KUKA KRL program: MyProgram_277().src

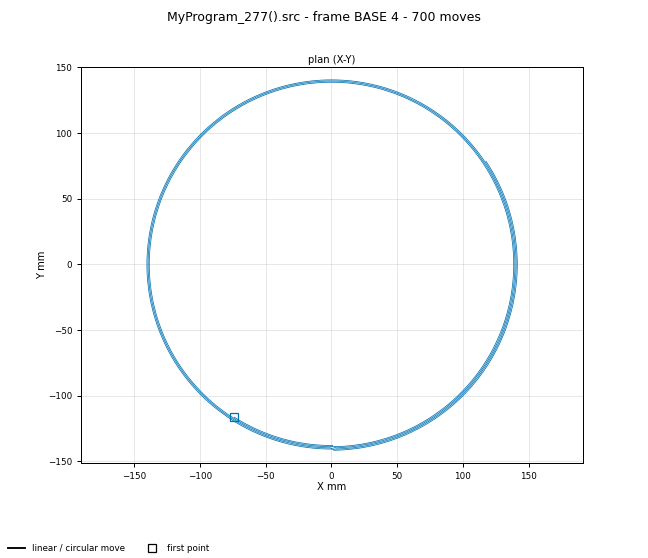
[picture p0: tool path of MyProgram_277().src in frame BASE 4, 700 of 700 moves have a stored position in this frame; points joined in program order, loops and branches not executed]
&ACCESS RVP
&REL 1
&PARAM TEMPLATE = C:\KRC\Roboter\Template\vorgabe
&PARAM EDITMASK = *
DEF MyProgram_277()
; ---- Setting reference (Base) ----
$BASE = BASE_DATA[4]

; --------------------------
; ---- Setting tool (TCP) ----
$TOOL = TOOL_DATA[3]
; --------------------------

$VEL.CP = VEL_APROX_PRINT
Startdeposition()
$VEL.CP = VEL_PRINT
LIN {X -74.0204,Y -116.2499,Z 172,A -119.7118,B 8.7917,C 0.3604,E1 8.715,E2 211.1655} C_DIS
LIN {X -70.2915,Y -118.5418,Z 172,A -117.8625,B 8.7917,C 0.3625,E1 8.7194,E2 209.3126} C_DIS
LIN {X -66.8151,Y -120.535,Z 172,A -115.8663,B 8.7917,C 0.3586,E1 8.7244,E2 207.2739} C_DIS
LIN {X -63.5094,Y -122.3084,Z 172,A -114.6724,B 8.7914,C 0.3673,E1 8.7272,E2 206.1271} C_DIS
LIN {X -60.8141,Y -123.6692,Z 172,A -113.4023,B 8.7914,C 0.3685,E1 8.7304,E2 204.8552} C_DIS
LIN {X -57.5799,Y -125.208,Z 172,A -111.8385,B 8.7914,C 0.3688,E1 8.7344,E2 203.2817} C_DIS
LIN {X -53.8139,Y -126.8742,Z 172,A -110.2313,B 8.7912,C 0.3725,E1 8.7385,E2 201.6879} C_DIS
LIN {X -51.2665,Y -127.9227,Z 172,A -109.0577,B 8.7912,C 0.3731,E1 8.7415,E2 200.5105} C_DIS
LIN {X -48.1192,Y -129.1395,Z 172,A -107.6615,B 8.7912,C 0.3745,E1 8.7452,E2 199.115} C_DIS
LIN {X -44.9658,Y -130.271,Z 172,A -106.2334,B 8.7912,C 0.375,E1 8.7489,E2 197.6822} C_DIS
LIN {X -41.408,Y -131.4462,Z 172,A -104.7037,B 8.791,C 0.3768,E1 8.753,E2 196.1559} C_DIS
LIN {X -38.8546,Y -132.2225,Z 172,A -103.5654,B 8.791,C 0.377,E1 8.7561,E2 195.0136} C_DIS
LIN {X -35.5653,Y -133.1449,Z 172,A -101.6158,B 8.7914,C 0.3678,E1 8.7615,E2 192.9952} C_DIS
LIN {X -31.1537,Y -134.2466,Z 172,A -100.099,B 8.7911,C 0.376,E1 8.7655,E2 191.5264} C_DIS
LIN {X -27.2255,Y -135.0974,Z 172,A -98.5166,B 8.791,C 0.3785,E1 8.7698,E2 189.9551} C_DIS
LIN {X -20.3148,Y -136.31,Z 172,A -95.7036,B 8.7908,C 0.3816,E1 8.7775,E2 187.1547} C_DIS
LIN {X -15.2753,Y -136.9652,Z 172,A -93.6377,B 8.7908,C 0.383,E1 8.7832,E2 185.0941} C_DIS
LIN {X -10.9275,Y -137.3811,Z 172,A -91.725,B 8.7908,C 0.3814,E1 8.7886,E2 183.1682} C_DIS
LIN {X -6.9698,Y -137.6371,Z 172,A -90.0219,B 8.7908,C 0.3804,E1 8.7933,E2 181.4573} C_DIS
LIN {X -2.6982,Y -137.7877,Z 172,A -88.2523,B 8.7908,C 0.3804,E1 8.7983,E2 179.688} C_DIS
LIN {X 0.9964,Y -137.8086,Z 172,A -86.8036,B 8.7908,C 0.382,E1 8.8023,E2 178.2498} C_DIS
Enddeposition()
LIN {X 0.9964,Y -137.8086,Z 172,A -86.8036,B 8.7908,C 0.382,E1 8.8023,E2 178.2498} C_DIS
Startdeposition()
$VEL.CP = VEL_PRINT
LIN {X 0.3242,Y -138.723,Z 172,A -87.6639,B 8.7185,C 0.4,E1 8.7281,E2 179.2402} C_DIS
LIN {X -3.8469,Y -138.6693,Z 172,A -89.329,B 8.7185,C 0.399,E1 8.7235,E2 180.8986} C_DIS
LIN {X -7.4248,Y -138.5245,Z 172,A -90.8807,B 8.7185,C 0.4004,E1 8.7191,E2 182.4603} C_DIS
LIN {X -11.8596,Y -138.2148,Z 172,A -92.6356,B 8.7185,C 0.3986,E1 8.7142,E2 184.2055} C_DIS
LIN {X -15.7064,Y -137.8324,Z 172,A -94.3982,B 8.7185,C 0.4015,E1 8.7093,E2 185.9901} C_DIS
LIN {X -20.165,Y -137.2501,Z 172,A -96.04,B 8.7187,C 0.3969,E1 8.7048,E2 187.6048} C_DIS
LIN {X -25.2134,Y -136.4125,Z 172,A -98.1321,B 8.7187,C 0.3957,E1 8.6991,E2 189.6948} C_DIS
LIN {X -28.3715,Y -135.792,Z 172,A -100.7545,B 8.7176,C 0.4193,E1 8.6915,E2 192.4824} C_DIS
LIN {X -36.4566,Y -133.8481,Z 172,A -102.9549,B 8.7188,C 0.3943,E1 8.6859,E2 194.5266} C_DIS
LIN {X -40.684,Y -132.6223,Z 172,A -104.8022,B 8.7188,C 0.3935,E1 8.681,E2 196.378} C_DIS
LIN {X -44.116,Y -131.5208,Z 172,A -106.2938,B 8.7188,C 0.3924,E1 8.677,E2 197.8702} C_DIS
LIN {X -47.3205,Y -130.402,Z 172,A -107.7112,B 8.7189,C 0.3915,E1 8.6733,E2 199.2898} C_DIS
LIN {X -50.4841,Y -129.2101,Z 172,A -109.1546,B 8.7189,C 0.3911,E1 8.6695,E2 200.7394} C_DIS
LIN {X -54.4235,Y -127.6024,Z 172,A -111.1054,B 8.7189,C 0.3928,E1 8.6644,E2 202.7151} C_DIS
LIN {X -58.4565,Y -125.8042,Z 172,A -112.7486,B 8.7191,C 0.3876,E1 8.6603,E2 204.3352} C_DIS
LIN {X -61.9898,Y -124.1029,Z 172,A -115.1913,B 8.7185,C 0.4004,E1 8.6539,E2 206.8828} C_DIS
LIN {X -67.5425,Y -121.1715,Z 172,A -117.0477,B 8.7192,C 0.384,E1 8.6496,E2 208.6456} C_DIS
LIN {X -71.4012,Y -118.9387,Z 172,A -118.9419,B 8.7193,C 0.3824,E1 8.645,E2 210.5464} C_DIS
LIN {X -75.2542,Y -116.5388,Z 172,A -120.8416,B 8.7194,C 0.3801,E1 8.6405,E2 212.4491} C_DIS
LIN {X -79.0577,Y -113.9925,Z 172,A -122.7073,B 8.7195,C 0.3767,E1 8.6362,E2 214.3114} C_DIS
LIN {X -84.8198,Y -109.7725,Z 172,A -125.6839,B 8.7197,C 0.3724,E1 8.6296,E2 217.2908} C_DIS
LIN {X -88.1962,Y -107.079,Z 172,A -127.5323,B 8.7198,C 0.3704,E1 8.6255,E2 219.1471} C_DIS
LIN {X -91.6854,Y -104.1068,Z 172,A -129.4351,B 8.72,C 0.3671,E1 8.6215,E2 221.0506} C_DIS
LIN {X -95.0471,Y -101.0467,Z 172,A -131.3319,B 8.72,C 0.3639,E1 8.6176,E2 222.9494} C_DIS
LIN {X -99.0959,Y -97.0792,Z 172,A -133.3125,B 8.7205,C 0.3531,E1 8.6138,E2 224.8833} C_DIS
LIN {X -104.511,Y -91.2239,Z 172,A -136.8158,B 8.7207,C 0.35,E1 8.6071,E2 228.4121} C_DIS
LIN {X -106.7656,Y -88.5747,Z 172,A -138.4803,B 8.7207,C 0.3507,E1 8.6041,E2 230.105} C_DIS
LIN {X -109.7218,Y -84.8852,Z 172,A -140.4212,B 8.7208,C 0.3462,E1 8.6007,E2 232.0436} C_DIS
LIN {X -112.3598,Y -81.3611,Z 172,A -142.2956,B 8.7209,C 0.343,E1 8.5976,E2 233.9243} C_DIS
LIN {X -115.06,Y -77.4962,Z 172,A -144.2731,B 8.7211,C 0.339,E1 8.5945,E2 235.9046} C_DIS
LIN {X -117.5369,Y -73.6859,Z 172,A -146.2134,B 8.7212,C 0.3355,E1 8.5915,E2 237.852} C_DIS
LIN {X -119.8595,Y -69.8443,Z 172,A -148.0404,B 8.7214,C 0.3306,E1 8.5889,E2 239.6745} C_DIS
LIN {X -122.1732,Y -65.7119,Z 172,A -150.0116,B 8.7216,C 0.3259,E1 8.5863,E2 241.6465} C_DIS
LIN {X -123.7944,Y -62.601,Z 172,A -151.3993,B 8.7217,C 0.3212,E1 8.5845,E2 243.0255} C_DIS
LIN {X -125.2991,Y -59.5317,Z 172,A -152.8494,B 8.7219,C 0.3182,E1 8.5828,E2 244.4795} C_DIS
LIN {X -126.7339,Y -56.4127,Z 172,A -154.3035,B 8.7219,C 0.3151,E1 8.5811,E2 245.9372} C_DIS
LIN {X -128.3144,Y -52.7245,Z 172,A -156.2703,B 8.7219,C 0.3158,E1 8.5789,E2 247.942} C_DIS
LIN {X -129.5181,Y -49.6916,Z 172,A -157.3054,B 8.7223,C 0.3072,E1 8.5779,E2 248.9368} C_DIS
LIN {X -131.4713,Y -44.2646,Z 172,A -159.609,B 8.7225,C 0.2995,E1 8.5758,E2 251.2287} C_DIS
LIN {X -132.7511,Y -40.2631,Z 172,A -161.5398,B 8.7225,C 0.2979,E1 8.5741,E2 253.183} C_DIS
LIN {X -133.6394,Y -37.2076,Z 172,A -162.8797,B 8.7227,C 0.2946,E1 8.5731,E2 254.5251} C_DIS
LIN {X -134.6865,Y -33.2261,Z 172,A -164.6911,B 8.7227,C 0.2917,E1 8.5719,E2 256.3492} C_DIS
LIN {X -135.5828,Y -29.3462,Z 172,A -166.2628,B 8.723,C 0.2859,E1 8.5709,E2 257.9104} C_DIS
LIN {X -136.2638,Y -26.0015,Z 172,A -167.6622,B 8.7231,C 0.2817,E1 8.5702,E2 259.3073} C_DIS
LIN {X -136.8367,Y -22.7954,Z 172,A -169.0722,B 8.7231,C 0.279,E1 8.5695,E2 260.7243} C_DIS
LIN {X -137.3787,Y -19.2651,Z 172,A -170.5699,B 8.7233,C 0.2751,E1 8.5689,E2 262.2236} C_DIS
LIN {X -137.8606,Y -15.4514,Z 172,A -172.6486,B 8.7233,C 0.2784,E1 8.5682,E2 264.3624} C_DIS
LIN {X -138.2652,Y -11.2629,Z 172,A -174.022,B 8.7235,C 0.2676,E1 8.5679,E2 265.6888} C_DIS
LIN {X -138.5435,Y -7.0462,Z 172,A -175.7765,B 8.7237,C 0.2627,E1 8.5676,E2 267.4428} C_DIS
LIN {X -138.711,Y -1.8533,Z 172,A -178.2848,B 8.7237,C 0.2622,E1 8.5674,E2 269.9944} C_DIS
LIN {X -138.7101,Y 1.9049,Z 172,A -179.3092,B 8.7241,C 0.2494,E1 8.5674,E2 270.9514} C_DIS
LIN {X -138.5749,Y 6.4229,Z 172,A 178.1704,B 8.7239,C 0.2543,E1 8.5677,E2 273.5516} C_DIS
LIN {X -138.3247,Y 10.5066,Z 172,A 176.9327,B 8.7243,C 0.2423,E1 8.568,E2 274.7315} C_DIS
LIN {X -137.8407,Y 15.6358,Z 172,A 174.7672,B 8.7244,C 0.2367,E1 8.5686,E2 276.8997} C_DIS
LIN {X -137.2685,Y 20.0363,Z 172,A 172.7833,B 8.7245,C 0.2338,E1 8.5693,E2 278.9006} C_DIS
LIN {X -136.4151,Y 25.2075,Z 172,A 170.1851,B 8.7245,C 0.2345,E1 8.5706,E2 281.5506} C_DIS
LIN {X -135.5943,Y 29.293,Z 172,A 168.916,B 8.7248,C 0.2224,E1 8.5713,E2 282.7618} C_DIS
LIN {X -134.8349,Y 32.6104,Z 172,A 167.4574,B 8.7248,C 0.2193,E1 8.5722,E2 284.2255} C_DIS
LIN {X -133.9949,Y 35.9063,Z 172,A 166.0442,B 8.725,C 0.2155,E1 8.5732,E2 285.6384} C_DIS
LIN {X -133.0835,Y 39.1493,Z 172,A 164.6359,B 8.725,C 0.2118,E1 8.5743,E2 287.0474} C_DIS
LIN {X -132.0225,Y 42.5917,Z 172,A 163.1561,B 8.7252,C 0.2076,E1 8.5756,E2 288.5247} C_DIS
LIN {X -131.0137,Y 45.5991,Z 172,A 161.7555,B 8.7252,C 0.2054,E1 8.5768,E2 289.9352} C_DIS
LIN {X -129.8339,Y 48.8574,Z 172,A 160.3395,B 8.7253,C 0.2013,E1 8.5782,E2 291.3479} C_DIS
LIN {X -128.5753,Y 52.0793,Z 172,A 158.8806,B 8.7253,C 0.1979,E1 8.5797,E2 292.809} C_DIS
LIN {X -127.2547,Y 55.2277,Z 172,A 157.4261,B 8.7255,C 0.1948,E1 8.5813,E2 294.2676} C_DIS
LIN {X -125.6381,Y 58.8157,Z 172,A 155.8229,B 8.7255,C 0.1901,E1 8.5832,E2 295.8665} C_DIS
LIN {X -124.2617,Y 61.6679,Z 172,A 154.4706,B 8.7256,C 0.1874,E1 8.5848,E2 297.2228} C_DIS
LIN {X -122.4601,Y 65.1761,Z 172,A 152.7126,B 8.7256,C 0.1853,E1 8.5871,E2 298.9953} C_DIS
LIN {X -119.3365,Y 70.7339,Z 172,A 150.1193,B 8.7258,C 0.178,E1 8.5907,E2 301.581} C_DIS
LIN {X -116.3027,Y 75.6178,Z 172,A 147.6553,B 8.7259,C 0.1735,E1 8.5944,E2 304.0536} C_DIS
LIN {X -113.6937,Y 79.487,Z 172,A 145.7234,B 8.7259,C 0.169,E1 8.5974,E2 305.984} C_DIS
LIN {X -111.1535,Y 83.0017,Z 172,A 143.496,B 8.7259,C 0.1718,E1 8.6012,E2 308.2634} C_DIS
LIN {X -108.5371,Y 86.3947,Z 172,A 142.3443,B 8.7262,C 0.1577,E1 8.6031,E2 309.3371} C_DIS
LIN {X -106.6108,Y 88.7617,Z 172,A 140.8413,B 8.7262,C 0.1588,E1 8.6058,E2 310.8689} C_DIS
LIN {X -103.3893,Y 92.4933,Z 172,A 138.5103,B 8.7262,C 0.1592,E1 8.6102,E2 313.2343} C_DIS
LIN {X -101.0197,Y 95.0758,Z 172,A 137.4276,B 8.7263,C 0.1501,E1 8.6121,E2 314.2705} C_DIS
LIN {X -98.3786,Y 97.806,Z 172,A 135.7273,B 8.7263,C 0.149,E1 8.6155,E2 315.9856} C_DIS
LIN {X -93.9427,Y 102.0741,Z 172,A 132.9381,B 8.7263,C 0.1479,E1 8.6212,E2 318.8028} C_DIS
LIN {X -91.5301,Y 104.2437,Z 172,A 131.8225,B 8.7265,C 0.1416,E1 8.6235,E2 319.8895} C_DIS
LIN {X -88.249,Y 107.0353,Z 172,A 129.9727,B 8.7265,C 0.1394,E1 8.6275,E2 321.7463} C_DIS
LIN {X -82.1585,Y 111.7781,Z 172,A 127.1438,B 8.7267,C 0.1277,E1 8.6336,E2 324.5279} C_DIS
LIN {X -78.0397,Y 114.6921,Z 172,A 124.603,B 8.7267,C 0.1319,E1 8.6395,E2 327.1233} C_DIS
LIN {X -73.0904,Y 117.9077,Z 172,A 122.4019,B 8.7267,C 0.124,E1 8.6446,E2 329.293} C_DIS
LIN {X -66.9602,Y 121.4939,Z 172,A 119.4226,B 8.7267,C 0.1205,E1 8.6519,E2 332.2757} C_DIS
LIN {X -63.9231,Y 123.118,Z 172,A 117.7393,B 8.7267,C 0.1231,E1 8.6561,E2 333.99} C_DIS
LIN {X -58.3449,Y 125.8558,Z 172,A 115.4948,B 8.7269,C 0.1142,E1 8.6616,E2 336.1927} C_DIS
LIN {X -55.4715,Y 127.1493,Z 172,A 113.9313,B 8.7269,C 0.1172,E1 8.6657,E2 337.7876} C_DIS
LIN {X -51.8822,Y 128.6548,Z 172,A 112.2929,B 8.7269,C 0.1159,E1 8.6699,E2 339.4284} C_DIS
LIN {X -46.991,Y 130.5208,Z 172,A 109.9792,B 8.7269,C 0.1164,E1 8.676,E2 341.7592} C_DIS
LIN {X -41.9253,Y 132.2354,Z 172,A 107.9603,B 8.7269,C 0.111,E1 8.6813,E2 343.7531} C_DIS
LIN {X -38.2224,Y 133.3549,Z 172,A 106.1871,B 8.7269,C 0.1128,E1 8.6861,E2 345.5468} C_DIS
LIN {X -33.626,Y 134.5861,Z 172,A 104.3973,B 8.7269,C 0.1081,E1 8.6909,E2 347.3137} C_DIS
LIN {X -30.0027,Y 135.441,Z 172,A 102.8676,B 8.7269,C 0.107,E1 8.6951,E2 348.8415} C_DIS
LIN {X -26.5988,Y 136.1496,Z 172,A 101.2804,B 8.7269,C 0.1089,E1 8.6994,E2 350.4464} C_DIS
LIN {X -21.2163,Y 137.0904,Z 172,A 99.0713,B 8.7269,C 0.1069,E1 8.7055,E2 352.6483} C_DIS
LIN {X -17.5847,Y 137.6041,Z 172,A 96.7454,B 8.7268,C 0.1211,E1 8.7123,E2 355.0724} C_DIS
LIN {X -11.1371,Y 138.2758,Z 172,A 95.0226,B 8.727,C 0.1028,E1 8.7167,E2 356.6771} C_DIS
LIN {X -5.0318,Y 138.6318,Z 172,A 92.3374,B 8.727,C 0.1054,E1 8.7242,E2 359.3807} C_DIS
LIN {X -0.8054,Y 138.7203,Z 172,A 90.5113,B 8.727,C 0.1068,E1 8.7294,E2 361.2159} C_DIS
LIN {X 4.2185,Y 138.6589,Z 172,A 88.0481,B 8.7269,C 0.1142,E1 8.7364,E2 363.7257} C_DIS
LIN {X 8.862,Y 138.4396,Z 172,A 86.6905,B 8.727,C 0.1038,E1 8.74,E2 365.0135} C_DIS
LIN {X 12.1595,Y 138.1894,Z 172,A 84.7302,B 8.7269,C 0.1154,E1 8.7456,E2 367.0464} C_DIS
LIN {X 16.9995,Y 137.6781,Z 172,A 83.1408,B 8.7269,C 0.1081,E1 8.7499,E2 368.5835} C_DIS
LIN {X 23.0161,Y 136.7998,Z 172,A 80.826,B 8.7269,C 0.1053,E1 8.7562,E2 370.8732} C_DIS
LIN {X 26.3072,Y 136.2053,Z 172,A 78.4486,B 8.7267,C 0.1253,E1 8.7631,E2 373.3724} C_DIS
LIN {X 33.2014,Y 134.6924,Z 172,A 76.5446,B 8.727,C 0.1076,E1 8.7679,E2 375.1519} C_DIS
LIN {X 37.2485,Y 133.6279,Z 172,A 74.7342,B 8.727,C 0.1105,E1 8.7728,E2 376.972} C_DIS
LIN {X 40.8786,Y 132.5627,Z 172,A 73.2457,B 8.727,C 0.1103,E1 8.7767,E2 378.4511} C_DIS
LIN {X 44.1498,Y 131.5095,Z 172,A 71.8406,B 8.727,C 0.1112,E1 8.7805,E2 379.8542} C_DIS
LIN {X 47.3458,Y 130.3929,Z 172,A 70.453,B 8.727,C 0.1124,E1 8.7841,E2 381.2403} C_DIS
LIN {X 50.2723,Y 129.2924,Z 172,A 69.1422,B 8.7269,C 0.1141,E1 8.7875,E2 382.5535} C_DIS
LIN {X 54.5821,Y 127.5338,Z 172,A 67.3645,B 8.7269,C 0.1132,E1 8.7921,E2 384.313} C_DIS
LIN {X 58.4211,Y 125.8206,Z 172,A 64.5472,B 8.7266,C 0.137,E1 8.7996,E2 387.2634} C_DIS
LIN {X 64.7088,Y 122.7054,Z 172,A 62.9534,B 8.7269,C 0.1144,E1 8.8031,E2 388.6964} C_DIS
LIN {X 67.2087,Y 121.3563,Z 172,A 61.3864,B 8.7267,C 0.1241,E1 8.8071,E2 390.3125} C_DIS
LIN {X 71.1242,Y 119.1039,Z 172,A 59.4228,B 8.7267,C 0.1288,E1 8.8118,E2 392.2884} C_DIS
LIN {X 75.3781,Y 116.4583,Z 172,A 57.4817,B 8.7267,C 0.1293,E1 8.8164,E2 394.2139} C_DIS
LIN {X 82.2077,Y 111.7419,Z 172,A 54.1644,B 8.7267,C 0.1327,E1 8.824,E2 397.5179} C_DIS
LIN {X 85.4379,Y 109.2924,Z 172,A 52.4373,B 8.7266,C 0.1367,E1 8.8278,E2 399.252} C_DIS
LIN {X 88.8891,Y 106.5046,Z 172,A 50.6069,B 8.7266,C 0.14,E1 8.8317,E2 401.0825} C_DIS
LIN {X 92.2706,Y 103.5888,Z 172,A 48.7975,B 8.7265,C 0.1427,E1 8.8355,E2 402.8881} C_DIS
LIN {X 95.7116,Y 100.4176,Z 172,A 47.0096,B 8.7265,C 0.1434,E1 8.8391,E2 404.6585} C_DIS
LIN {X 98.382,Y 97.8025,Z 172,A 45.1328,B 8.7263,C 0.1536,E1 8.8429,E2 406.5773} C_DIS
LIN {X 100.7828,Y 95.3268,Z 172,A 43.6912,B 8.7263,C 0.1569,E1 8.8457,E2 408.0216} C_DIS
LIN {X 103.2399,Y 92.6601,Z 172,A 42.6367,B 8.7263,C 0.1507,E1 8.8476,E2 409.0214} C_DIS
LIN {X 105.6518,Y 89.9002,Z 172,A 40.9694,B 8.7263,C 0.1573,E1 8.8507,E2 410.7085} C_DIS
LIN {X 108.5223,Y 86.4134,Z 172,A 39.1254,B 8.7261,C 0.161,E1 8.8539,E2 412.5506} C_DIS
LIN {X 111.37,Y 82.711,Z 172,A 37.2314,B 8.7261,C 0.1646,E1 8.8571,E2 414.441} C_DIS
LIN {X 113.9088,Y 79.1779,Z 172,A 35.409,B 8.726,C 0.1694,E1 8.86,E2 416.2675} C_DIS
LIN {X 116.2608,Y 75.6824,Z 172,A 33.716,B 8.726,C 0.1725,E1 8.8626,E2 417.9555} C_DIS
LIN {X 119.9112,Y 69.7549,Z 172,A 30.9127,B 8.7258,C 0.1781,E1 8.8667,E2 420.7514} C_DIS
LIN {X 122.0614,Y 65.9201,Z 172,A 29.1131,B 8.7258,C 0.1823,E1 8.8691,E2 422.55} C_DIS
LIN {X 123.7718,Y 62.6454,Z 172,A 27.6566,B 8.7257,C 0.1846,E1 8.8709,E2 423.9987} C_DIS
LIN {X 125.8051,Y 58.4547,Z 172,A 26.0177,B 8.7257,C 0.1834,E1 8.8729,E2 425.6028} C_DIS
LIN {X 127.2304,Y 55.2838,Z 172,A 23.9557,B 8.7253,C 0.2009,E1 8.8753,E2 427.7445} C_DIS
LIN {X 128.8371,Y 51.4299,Z 172,A 22.7158,B 8.7255,C 0.1949,E1 8.8765,E2 428.9247} C_DIS
LIN {X 130.04,Y 48.307,Z 172,A 21.3959,B 8.7255,C 0.1972,E1 8.8778,E2 430.2378} C_DIS
LIN {X 131.0721,Y 45.4306,Z 172,A 20.0472,B 8.7253,C 0.2026,E1 8.8791,E2 431.5983} C_DIS
LIN {X 132.3723,Y 41.4968,Z 172,A 18.272,B 8.7251,C 0.2087,E1 8.8806,E2 433.3829} C_DIS
LIN {X 133.5512,Y 37.5228,Z 172,A 16.7028,B 8.7251,C 0.2103,E1 8.8818,E2 434.9353} C_DIS
LIN {X 134.4535,Y 34.1486,Z 172,A 15.2678,B 8.7251,C 0.2141,E1 8.8828,E2 436.3704} C_DIS
LIN {X 135.237,Y 30.9004,Z 172,A 13.4585,B 8.7247,C 0.2275,E1 8.884,E2 438.2349} C_DIS
LIN {X 136.1633,Y 26.527,Z 172,A 12.2619,B 8.7249,C 0.2183,E1 8.8846,E2 439.3511} C_DIS
LIN {X 136.8857,Y 22.5014,Z 172,A 10.4407,B 8.7247,C 0.2261,E1 8.8855,E2 441.1904} C_DIS
LIN {X 137.4958,Y 18.411,Z 172,A 8.085,B 8.7242,C 0.2453,E1 8.8864,E2 443.6291} C_DIS
LIN {X 138.1289,Y 12.8265,Z 172,A 6.5251,B 8.7245,C 0.2351,E1 8.8868,E2 445.0951} C_DIS
LIN {X 138.433,Y 8.9691,Z 172,A 4.3499,B 8.724,C 0.2526,E1 8.8873,E2 447.3446} C_DIS
LIN {X 138.6635,Y 4.0543,Z 172,A 2.4626,B 8.724,C 0.2553,E1 8.8874,E2 449.2155} C_DIS
LIN {X 138.7241,Y -0.3949,Z 172,A 1.0019,B 8.724,C 0.2522,E1 8.8874,E2 450.6303} C_DIS
LIN {X 138.6599,Y -4.1841,Z 172,A -0.9485,B 8.7236,C 0.2653,E1 8.8873,E2 452.6309} C_DIS
LIN {X 138.4392,Y -8.8691,Z 172,A -2.2659,B 8.7239,C 0.2571,E1 8.8871,E2 453.8716} C_DIS
LIN {X 137.865,Y -15.4112,Z 172,A -4.9417,B 8.7237,C 0.2642,E1 8.8864,E2 456.5454} C_DIS
LIN {X 137.4428,Y -18.815,Z 172,A -6.6169,B 8.7233,C 0.274,E1 8.8857,E2 458.255} C_DIS
LIN {X 136.6846,Y -23.7013,Z 172,A -8.9308,B 8.723,C 0.286,E1 8.8847,E2 460.6053} C_DIS
LIN {X 135.7985,Y -28.3394,Z 172,A -10.1846,B 8.7233,C 0.276,E1 8.884,E2 461.7725} C_DIS
LIN {X 134.7881,Y -32.8043,Z 172,A -12.1615,B 8.7231,C 0.2833,E1 8.8827,E2 463.7623} C_DIS
LIN {X 133.7501,Y -36.8118,Z 172,A -14.229,B 8.7226,C 0.2961,E1 8.8812,E2 465.8771} C_DIS
LIN {X 132.7031,Y -40.4198,Z 172,A -15.1321,B 8.723,C 0.286,E1 8.8806,E2 466.6989} C_DIS
LIN {X 131.5159,Y -44.1307,Z 172,A -16.9973,B 8.7226,C 0.2962,E1 8.8789,E2 468.5986} C_DIS
LIN {X 130.1884,Y -47.9108,Z 172,A -19.1411,B 8.7221,C 0.3116,E1 8.8768,E2 470.8065} C_DIS
LIN {X 128.4857,Y -52.3016,Z 172,A -20.3259,B 8.7225,C 0.3,E1 8.8757,E2 471.8963} C_DIS
LIN {X 124.6131,Y -60.9555,Z 172,A -24.2138,B 8.7222,C 0.31,E1 8.8713,E2 475.785} C_DIS
LIN {X 122.9685,Y -64.2078,Z 172,A -25.7889,B 8.722,C 0.3155,E1 8.8692,E2 477.3706} C_DIS
LIN {X 121.1051,Y -67.6612,Z 172,A -27.5027,B 8.7217,C 0.3217,E1 8.8669,E2 479.0981} C_DIS
LIN {X 119.0443,Y -71.2241,Z 172,A -29.2756,B 8.7215,C 0.3277,E1 8.8644,E2 480.8821} C_DIS
LIN {X 115.8531,Y -76.3048,Z 172,A -31.4493,B 8.7215,C 0.3271,E1 8.8612,E2 483.0192} C_DIS
LIN {X 113.9507,Y -79.1177,Z 172,A -32.9952,B 8.7213,C 0.3337,E1 8.8587,E2 484.585} C_DIS
LIN {X 111.152,Y -83.0038,Z 172,A -35.2261,B 8.7209,C 0.344,E1 8.8549,E2 486.8504} C_DIS
LIN {X 108.9602,Y -85.8608,Z 172,A -36.3984,B 8.721,C 0.3406,E1 8.853,E2 487.9839} C_DIS
LIN {X 107.0456,Y -88.2366,Z 172,A -38.2917,B 8.7204,C 0.3573,E1 8.8495,E2 489.9595} C_DIS
LIN {X 103.4304,Y -92.4474,Z 172,A -39.8345,B 8.7208,C 0.3462,E1 8.8468,E2 491.4087} C_DIS
LIN {X 98.7972,Y -97.3837,Z 172,A -42.5813,B 8.7206,C 0.3512,E1 8.8415,E2 494.1521} C_DIS
LIN {X 96.1623,Y -99.9868,Z 172,A -44.4067,B 8.7202,C 0.3608,E1 8.8378,E2 496.0169} C_DIS
LIN {X 92.4449,Y -103.4327,Z 172,A -46.8779,B 8.7197,C 0.3732,E1 8.8326,E2 498.5385} C_DIS
LIN {X 88.2994,Y -106.9936,Z 172,A -48.4863,B 8.7201,C 0.3637,E1 8.8293,E2 500.066} C_DIS
LIN {X 84.3762,Y -110.1137,Z 172,A -50.6802,B 8.7198,C 0.3702,E1 8.8244,E2 502.2777} C_DIS
LIN {X 78.3351,Y -114.4902,Z 172,A -53.6127,B 8.7198,C 0.3725,E1 8.8178,E2 505.194} C_DIS
LIN {X 74.5642,Y -116.9812,Z 172,A -56.1261,B 8.719,C 0.3893,E1 8.8117,E2 507.7919} C_DIS
LIN {X 69.5847,Y -120.0097,Z 172,A -57.8224,B 8.7195,C 0.3781,E1 8.8078,E2 509.3993} C_DIS
LIN {X 65.9915,Y -122.0231,Z 172,A -59.5568,B 8.7193,C 0.3813,E1 8.8035,E2 511.1395} C_DIS
LIN {X 62.6783,Y -123.755,Z 172,A -61.0237,B 8.7193,C 0.3819,E1 8.7999,E2 512.5976} C_DIS
LIN {X 59.2574,Y -125.4302,Z 172,A -62.5435,B 8.7193,C 0.3829,E1 8.7961,E2 514.1118} C_DIS
LIN {X 55.2623,Y -127.2397,Z 172,A -64.4194,B 8.7191,C 0.3866,E1 8.7913,E2 515.9975} C_DIS
LIN {X 51.8854,Y -128.6535,Z 172,A -65.8213,B 8.7191,C 0.3862,E1 8.7877,E2 517.3864} C_DIS
LIN {X 47.4409,Y -130.3586,Z 172,A -67.9658,B 8.7189,C 0.3921,E1 8.782,E2 519.5554} C_DIS
LIN {X 41.791,Y -132.2783,Z 172,A -70.2008,B 8.7189,C 0.3899,E1 8.7762,E2 521.7626} C_DIS
LIN {X 38.6297,Y -133.2356,Z 172,A -71.6202,B 8.7189,C 0.3923,E1 8.7724,E2 523.1901} C_DIS
LIN {X 35.34,Y -134.1459,Z 172,A -73.593,B 8.7183,C 0.4049,E1 8.7669,E2 525.2362} C_DIS
LIN {X 30.541,Y -135.3191,Z 172,A -75.1325,B 8.7187,C 0.3964,E1 8.7628,E2 526.7129} C_DIS
LIN {X 26.2684,Y -136.2127,Z 172,A -77.1393,B 8.7184,C 0.4017,E1 8.7573,E2 528.7471} C_DIS
LIN {X 22.9255,Y -136.815,Z 172,A -78.1261,B 8.7188,C 0.3942,E1 8.7547,E2 529.6812} C_DIS
LIN {X 16.3705,Y -137.7531,Z 172,A -80.9476,B 8.7186,C 0.3974,E1 8.7468,E2 532.5155} C_DIS
LIN {X 12.5483,Y -138.1556,Z 172,A -82.7068,B 8.7185,C 0.4015,E1 8.7419,E2 534.2979} C_DIS
LIN {X 8.2908,Y -138.4748,Z 172,A -84.3314,B 8.7185,C 0.3993,E1 8.7374,E2 535.9055} C_DIS
LIN {X 4.1301,Y -138.6614,Z 172,A -86.0461,B 8.7185,C 0.3996,E1 8.7326,E2 537.6204} C_DIS
LIN {X 1.0053,Y -138.7163,Z 172,A -86.8635,B 8.7189,C 0.3904,E1 8.7305,E2 538.377} C_DIS
Enddeposition()
LIN {X 1.0053,Y -138.7163,Z 172,A -86.8635,B 8.7189,C 0.3904,E1 8.7305,E2 538.377} C_DIS
Startdeposition()
$VEL.CP = VEL_PRINT
LIN {X 3.4172,Y -139.5907,Z 172,A -85.4867,B 8.4576,C 0.3922,E1 8.4731,E2 537.0591} C_DIS
LIN {X 7.4799,Y -139.432,Z 172,A -83.9285,B 8.4576,C 0.3939,E1 8.4774,E2 535.5145} C_DIS
LIN {X 11.4262,Y -139.1638,Z 172,A -82.3394,B 8.4575,C 0.394,E1 8.4819,E2 533.929} C_DIS
LIN {X 14.5932,Y -138.8674,Z 172,A -81.0545,B 8.4575,C 0.3939,E1 8.4854,E2 532.646} C_DIS
LIN {X 17.041,Y -138.5888,Z 172,A -79.6692,B 8.4579,C 0.386,E1 8.4894,E2 531.2108} C_DIS
LIN {X 20.4055,Y -138.1334,Z 172,A -78.347,B 8.4579,C 0.3866,E1 8.493,E2 529.8971} C_DIS
LIN {X 28.6687,Y -136.6591,Z 172,A -75.169,B 8.4577,C 0.3897,E1 8.5017,E2 526.7522} C_DIS
LIN {X 36.0489,Y -134.8978,Z 172,A -72.0226,B 8.4578,C 0.3866,E1 8.5102,E2 523.5995} C_DIS
LIN {X 40.2023,Y -133.7205,Z 172,A -70.216,B 8.4579,C 0.3842,E1 8.5151,E2 521.7871} C_DIS
LIN {X 47.5147,Y -131.2984,Z 172,A -67.1029,B 8.458,C 0.3819,E1 8.5233,E2 518.6779} C_DIS
LIN {X 51.3152,Y -129.8624,Z 172,A -65.3647,B 8.4582,C 0.3785,E1 8.5278,E2 516.9291} C_DIS
LIN {X 57.8623,Y -127.0794,Z 172,A -62.5187,B 8.4582,C 0.3764,E1 8.5351,E2 514.0905} C_DIS
LIN {X 61.4553,Y -125.3804,Z 172,A -60.9254,B 8.4584,C 0.3749,E1 8.5391,E2 512.5007} C_DIS
LIN {X 64.6852,Y -123.7447,Z 172,A -59.519,B 8.4584,C 0.3745,E1 8.5426,E2 511.1036} C_DIS
LIN {X 68.4312,Y -121.7153,Z 172,A -57.6469,B 8.4586,C 0.3692,E1 8.5472,E2 509.2137} C_DIS
LIN {X 73.7615,Y -118.5604,Z 172,A -54.9381,B 8.4589,C 0.3617,E1 8.5537,E2 506.4806} C_DIS
LIN {X 76.7311,Y -116.6609,Z 172,A -53.891,B 8.4587,C 0.3677,E1 8.5561,E2 505.4848} C_DIS
LIN {X 79.9554,Y -114.4749,Z 172,A -52.1056,B 8.459,C 0.3609,E1 8.5602,E2 503.6734} C_DIS
LIN {X 84.0164,Y -111.5289,Z 172,A -50.1214,B 8.459,C 0.3588,E1 8.5647,E2 501.6972} C_DIS
LIN {X 87.537,Y -108.7875,Z 172,A -48.3154,B 8.4592,C 0.3559,E1 8.5686,E2 499.8927} C_DIS
LIN {X 92.3457,Y -104.7364,Z 172,A -45.5787,B 8.4595,C 0.3474,E1 8.5745,E2 497.1329} C_DIS
LIN {X 94.7501,Y -102.5669,Z 172,A -44.4555,B 8.4595,C 0.3492,E1 8.5767,E2 496.0356} C_DIS
LIN {X 97.9718,Y -99.4939,Z 172,A -42.6266,B 8.4596,C 0.3453,E1 8.5804,E2 494.2046} C_DIS
LIN {X 102.2649,Y -95.0754,Z 172,A -39.9497,B 8.46,C 0.3366,E1 8.5856,E2 491.5056} C_DIS
LIN {X 104.4899,Y -92.6247,Z 172,A -38.7922,B 8.46,C 0.3379,E1 8.5877,E2 490.3732} C_DIS
LIN {X 107.3706,Y -89.2696,Z 172,A -37.0224,B 8.46,C 0.3347,E1 8.5909,E2 488.6074} C_DIS
LIN {X 112.1616,Y -83.1702,Z 172,A -33.9043,B 8.4603,C 0.3287,E1 8.5962,E2 485.4947} C_DIS
LIN {X 115.1513,Y -78.9785,Z 172,A -31.7915,B 8.4605,C 0.3236,E1 8.5996,E2 483.3798} C_DIS
LIN {X 117.5025,Y -75.4357,Z 172,A -29.8969,B 8.4608,C 0.3159,E1 8.6025,E2 481.4637} C_DIS
LIN {X 119.2361,Y -72.666,Z 172,A -28.7233,B 8.4608,C 0.3162,E1 8.6042,E2 480.3107} C_DIS
LIN {X 121.3286,Y -69.1146,Z 172,A -27.0922,B 8.4608,C 0.3132,E1 8.6064,E2 478.6857} C_DIS
LIN {X 123.455,Y -65.2368,Z 172,A -25.3619,B 8.461,C 0.3104,E1 8.6087,E2 476.9646} C_DIS
LIN {X 125.6824,Y -60.8385,Z 172,A -22.724,B 8.4616,C 0.2914,E1 8.6121,E2 474.2438} C_DIS
LIN {X 127.9588,Y -55.8901,Z 172,A -21.153,B 8.4613,C 0.3002,E1 8.6137,E2 472.7579} C_DIS
LIN {X 129.397,Y -52.4726,Z 172,A -19.7569,B 8.4613,C 0.2988,E1 8.6152,E2 471.3765} C_DIS
LIN {X 131.1253,Y -47.9949,Z 172,A -17.631,B 8.4617,C 0.29,E1 8.6173,E2 469.2283} C_DIS
LIN {X 132.3889,Y -44.3865,Z 172,A -16.2099,B 8.4617,C 0.2889,E1 8.6186,E2 467.8249} C_DIS
LIN {X 133.402,Y -41.243,Z 172,A -14.8134,B 8.4619,C 0.2842,E1 8.6198,E2 466.4216} C_DIS
LIN {X 134.9035,Y -36.0273,Z 172,A -12.9836,B 8.4618,C 0.2867,E1 8.6211,E2 464.6413} C_DIS
LIN {X 135.9716,Y -31.7671,Z 172,A -10.8384,B 8.4622,C 0.2741,E1 8.6226,E2 462.4498} C_DIS
LIN {X 137.1236,Y -26.3458,Z 172,A -8.6886,B 8.4623,C 0.2703,E1 8.6238,E2 460.314} C_DIS
LIN {X 137.8574,Y -22.202,Z 172,A -6.934,B 8.4625,C 0.2648,E1 8.6246,E2 458.5542} C_DIS
LIN {X 138.3919,Y -18.5701,Z 172,A -5.5023,B 8.4625,C 0.2621,E1 8.6251,E2 457.1306} C_DIS
LIN {X 138.8979,Y -14.3099,Z 172,A -3.4697,B 8.4629,C 0.2509,E1 8.6258,E2 455.0609} C_DIS
LIN {X 139.2107,Y -10.8556,Z 172,A -2.3153,B 8.4629,C 0.2528,E1 8.626,E2 453.9402} C_DIS
LIN {X 139.5243,Y -5.4766,Z 172,A -0.1392,B 8.463,C 0.2472,E1 8.6263,E2 451.7666} C_DIS
LIN {X 139.6263,Y -1.4101,Z 172,A 1.3867,B 8.463,C 0.2455,E1 8.6264,E2 450.2578} C_DIS
LIN {X 139.5844,Y 3.6429,Z 172,A 3.7846,B 8.4634,C 0.2323,E1 8.6263,E2 447.8158} C_DIS
LIN {X 139.4516,Y 7.0914,Z 172,A 4.8903,B 8.4634,C 0.2351,E1 8.6261,E2 446.7493} C_DIS
LIN {X 139.1746,Y 11.2977,Z 172,A 6.521,B 8.4634,C 0.2323,E1 8.6258,E2 445.1298} C_DIS
LIN {X 138.9535,Y 13.7508,Z 172,A 7.9048,B 8.4637,C 0.2211,E1 8.6254,E2 443.6968} C_DIS
LIN {X 138.5368,Y 17.4643,Z 172,A 9.2268,B 8.4637,C 0.2214,E1 8.625,E2 442.401} C_DIS
LIN {X 137.2757,Y 25.5499,Z 172,A 12.3044,B 8.4638,C 0.2181,E1 8.6236,E2 439.357} C_DIS
LIN {X 135.8494,Y 32.2814,Z 172,A 15.1955,B 8.4641,C 0.2087,E1 8.6219,E2 436.4551} C_DIS
LIN {X 134.9571,Y 35.8265,Z 172,A 16.6381,B 8.4641,C 0.2057,E1 8.6209,E2 435.0188} C_DIS
LIN {X 134.0992,Y 38.9158,Z 172,A 17.8979,B 8.4641,C 0.2033,E1 8.6199,E2 433.7651} C_DIS
LIN {X 133.0705,Y 42.2989,Z 172,A 19.4024,B 8.4643,C 0.1982,E1 8.6187,E2 432.2527} C_DIS
LIN {X 131.825,Y 46.0344,Z 172,A 20.9519,B 8.4643,C 0.1952,E1 8.6173,E2 430.7106} C_DIS
LIN {X 130.3096,Y 50.1648,Z 172,A 22.7155,B 8.4645,C 0.1913,E1 8.6155,E2 428.9511} C_DIS
LIN {X 127.8422,Y 56.1585,Z 172,A 25.3684,B 8.4646,C 0.1844,E1 8.6127,E2 426.2974} C_DIS
LIN {X 126.6874,Y 58.7127,Z 172,A 26.6006,B 8.4647,C 0.1796,E1 8.6112,E2 425.0539} C_DIS
LIN {X 124.6025,Y 63.0176,Z 172,A 28.4075,B 8.4647,C 0.1779,E1 8.609,E2 423.2659} C_DIS
LIN {X 122.8012,Y 66.4641,Z 172,A 30.0743,B 8.4649,C 0.1723,E1 8.6068,E2 421.5891} C_DIS
LIN {X 120.7527,Y 70.116,Z 172,A 31.9958,B 8.465,C 0.1637,E1 8.6041,E2 419.6405} C_DIS
LIN {X 118.9079,Y 73.2003,Z 172,A 33.3022,B 8.465,C 0.1637,E1 8.6022,E2 418.3549} C_DIS
LIN {X 116.1723,Y 77.4689,Z 172,A 35.2811,B 8.465,C 0.1609,E1 8.5992,E2 416.3881} C_DIS
LIN {X 113.403,Y 81.4695,Z 172,A 37.2375,B 8.4652,C 0.1571,E1 8.5961,E2 414.4359} C_DIS
LIN {X 111.0202,Y 84.6875,Z 172,A 38.6812,B 8.4652,C 0.1575,E1 8.5937,E2 413.0169} C_DIS
LIN {X 108.7547,Y 87.5776,Z 172,A 40.3302,B 8.4652,C 0.1511,E1 8.5908,E2 411.3491} C_DIS
LIN {X 105.9495,Y 90.9516,Z 172,A 42.1069,B 8.4653,C 0.1477,E1 8.5876,E2 409.5747} C_DIS
LIN {X 101.2929,Y 96.111,Z 172,A 44.9408,B 8.4654,C 0.1421,E1 8.5822,E2 406.7422} C_DIS
LIN {X 97.8695,Y 99.5942,Z 172,A 46.7507,B 8.4654,C 0.1421,E1 8.5787,E2 404.9564} C_DIS
LIN {X 95.3209,Y 102.0363,Z 172,A 48.4034,B 8.4655,C 0.135,E1 8.5753,E2 403.2772} C_DIS
LIN {X 91.5925,Y 105.396,Z 172,A 50.37,B 8.4655,C 0.133,E1 8.5712,E2 401.322} C_DIS
LIN {X 88.2208,Y 108.2338,Z 172,A 52.1545,B 8.4656,C 0.1302,E1 8.5674,E2 399.5401} C_DIS
LIN {X 84.5859,Y 111.0979,Z 172,A 54.0179,B 8.4656,C 0.1276,E1 8.5633,E2 397.6808} C_DIS
LIN {X 77.5197,Y 116.1384,Z 172,A 57.6525,B 8.4658,C 0.1203,E1 8.5549,E2 394.0366} C_DIS
LIN {X 73.8455,Y 118.5086,Z 172,A 59.4178,B 8.4658,C 0.1181,E1 8.5508,E2 392.2748} C_DIS
LIN {X 69.5523,Y 121.0788,Z 172,A 61.4202,B 8.4658,C 0.1162,E1 8.546,E2 390.2787} C_DIS
LIN {X 65.6231,Y 123.2522,Z 172,A 63.165,B 8.4658,C 0.1157,E1 8.5417,E2 388.5463} C_DIS
LIN {X 56.8088,Y 127.5527,Z 172,A 67.5213,B 8.466,C 0.1041,E1 8.5306,E2 384.148} C_DIS
LIN {X 52.9844,Y 129.1907,Z 172,A 68.8901,B 8.466,C 0.109,E1 8.5272,E2 382.8225} C_DIS
LIN {X 49.3386,Y 130.6244,Z 172,A 70.4224,B 8.466,C 0.1088,E1 8.5232,E2 381.2998} C_DIS
LIN {X 46.0081,Y 131.8341,Z 172,A 71.876,B 8.466,C 0.1075,E1 8.5194,E2 379.8464} C_DIS
LIN {X 43.0285,Y 132.8374,Z 172,A 73.1984,B 8.466,C 0.1057,E1 8.5159,E2 378.5202} C_DIS
LIN {X 39.4683,Y 133.9374,Z 172,A 74.6505,B 8.466,C 0.1059,E1 8.512,E2 377.078} C_DIS
LIN {X 35.9947,Y 134.9122,Z 172,A 76.1238,B 8.466,C 0.105,E1 8.5081,E2 375.6059} C_DIS
LIN {X 32.2813,Y 135.8494,Z 172,A 78.806,B 8.4662,C 0.0823,E1 8.5004,E2 372.7825} C_DIS
LIN {X 24.6028,Y 137.4469,Z 172,A 80.5894,B 8.4659,C 0.1084,E1 8.496,E2 371.1827} C_DIS
LIN {X 19.2773,Y 138.2953,Z 172,A 83.1849,B 8.466,C 0.1002,E1 8.4887,E2 368.5399} C_DIS
LIN {X 13.9108,Y 138.9382,Z 172,A 85.3878,B 8.466,C 0.0998,E1 8.4826,E2 366.3396} C_DIS
LIN {X 10.0951,Y 139.2663,Z 172,A 86.9067,B 8.466,C 0.1004,E1 8.4784,E2 364.8279} C_DIS
LIN {X 5.1289,Y 139.5379,Z 172,A 89.1857,B 8.466,C 0.0957,E1 8.4719,E2 362.5197} C_DIS
LIN {X -0.2934,Y 139.6323,Z 172,A 91.2188,B 8.466,C 0.0993,E1 8.4663,E2 360.5119} C_DIS
LIN {X -4.3706,Y 139.5642,Z 172,A 92.7803,B 8.466,C 0.1015,E1 8.462,E2 358.9653} C_DIS
LIN {X -9.086,Y 139.3367,Z 172,A 94.7582,B 8.466,C 0.1011,E1 8.4565,E2 356.9832} C_DIS
LIN {X -15.3218,Y 138.789,Z 172,A 97.4467,B 8.466,C 0.0996,E1 8.449,E2 354.2811} C_DIS
LIN {X -19.5532,Y 138.2559,Z 172,A 99.8422,B 8.4661,C 0.0886,E1 8.4421,E2 351.8047} C_DIS
LIN {X -25.3755,Y 137.3086,Z 172,A 101.8792,B 8.4661,C 0.0968,E1 8.4367,E2 349.8181} C_DIS
LIN {X -28.8894,Y 136.6115,Z 172,A 103.0997,B 8.466,C 0.1022,E1 8.4334,E2 348.63} C_DIS
LIN {X -32.5283,Y 135.7899,Z 172,A 104.5602,B 8.466,C 0.1045,E1 8.4295,E2 347.1792} C_DIS
LIN {X -36.8029,Y 134.6966,Z 172,A 106.5044,B 8.466,C 0.1035,E1 8.4242,E2 345.2195} C_DIS
LIN {X -40.3622,Y 133.6716,Z 172,A 107.8994,B 8.466,C 0.107,E1 8.4205,E2 343.8413} C_DIS
LIN {X -43.8275,Y 132.5751,Z 172,A 109.5413,B 8.466,C 0.1057,E1 8.4161,E2 342.1814} C_DIS
LIN {X -50.0911,Y 130.3382,Z 172,A 112.2883,B 8.466,C 0.1082,E1 8.4089,E2 339.4343} C_DIS
LIN {X -54.8521,Y 128.4076,Z 172,A 114.2371,B 8.4659,C 0.1133,E1 8.4039,E2 337.5072} C_DIS
LIN {X -57.7884,Y 127.1136,Z 172,A 115.9734,B 8.4659,C 0.1076,E1 8.3994,E2 335.7189} C_DIS
LIN {X -61.2524,Y 125.4805,Z 172,A 117.2268,B 8.4659,C 0.1151,E1 8.3963,E2 334.5069} C_DIS
LIN {X -64.6364,Y 123.7703,Z 172,A 118.7392,B 8.4658,C 0.1179,E1 8.3926,E2 333.0013} C_DIS
LIN {X -67.4703,Y 122.2507,Z 172,A 120.686,B 8.4659,C 0.1091,E1 8.3876,E2 330.9763} C_DIS
LIN {X -71.9259,Y 119.6839,Z 172,A 122.3191,B 8.4658,C 0.1204,E1 8.3839,E2 329.4055} C_DIS
LIN {X -76.9556,Y 116.5131,Z 172,A 124.7524,B 8.4657,C 0.1244,E1 8.3782,E2 326.9751} C_DIS
LIN {X -80.6289,Y 114.0019,Z 172,A 126.4552,B 8.4657,C 0.1295,E1 8.3743,E2 325.2895} C_DIS
LIN {X -82.9982,Y 112.2892,Z 172,A 127.791,B 8.4657,C 0.1293,E1 8.3712,E2 323.9375} C_DIS
LIN {X -88.3791,Y 108.1044,Z 172,A 130.6154,B 8.4656,C 0.1339,E1 8.3651,E2 321.1124} C_DIS
LIN {X -91.1413,Y 105.7861,Z 172,A 132.6056,B 8.4656,C 0.1282,E1 8.3607,E2 319.0589} C_DIS
LIN {X -94.7517,Y 102.5654,Z 172,A 134.7616,B 8.4656,C 0.1293,E1 8.3562,E2 316.883} C_DIS
LIN {X -98.7966,Y 98.6752,Z 172,A 136.5063,B 8.4654,C 0.1433,E1 8.3529,E2 315.2114} C_DIS
LIN {X -104.2978,Y 92.8416,Z 172,A 140.2181,B 8.4654,C 0.1435,E1 8.3458,E2 311.4495} C_DIS
LIN {X -107.213,Y 89.4591,Z 172,A 141.6601,B 8.4652,C 0.1539,E1 8.3433,E2 310.0588} C_DIS
LIN {X -109.1629,Y 87.0684,Z 172,A 143.1205,B 8.4652,C 0.1537,E1 8.3407,E2 308.5751} C_DIS
LIN {X -111.1409,Y 84.5297,Z 172,A 144.2762,B 8.4652,C 0.1594,E1 8.3388,E2 307.4415} C_DIS
LIN {X -113.8275,Y 80.8758,Z 172,A 146.1792,B 8.465,C 0.1631,E1 8.3357,E2 305.5351} C_DIS
LIN {X -116.3679,Y 77.1759,Z 172,A 147.9097,B 8.465,C 0.1694,E1 8.333,E2 303.8205} C_DIS
LIN {X -118.6511,Y 73.616,Z 172,A 149.9164,B 8.465,C 0.1693,E1 8.33,E2 301.7811} C_DIS
LIN {X -121.148,Y 69.431,Z 172,A 151.9372,B 8.4648,C 0.174,E1 8.3271,E2 299.7597} C_DIS
LIN {X -123.4571,Y 65.233,Z 172,A 153.7535,B 8.4647,C 0.1814,E1 8.3248,E2 297.9643} C_DIS
LIN {X -125.0524,Y 62.1201,Z 172,A 155.1958,B 8.4646,C 0.185,E1 8.3229,E2 296.5226} C_DIS
LIN {X -126.5947,Y 58.9133,Z 172,A 156.684,B 8.4646,C 0.1884,E1 8.3212,E2 295.0324} C_DIS
LIN {X -128.0201,Y 55.7483,Z 172,A 158.0418,B 8.4644,C 0.1933,E1 8.3196,E2 293.6844} C_DIS
LIN {X -129.3948,Y 52.4782,Z 172,A 159.5938,B 8.4644,C 0.1957,E1 8.318,E2 292.1216} C_DIS
LIN {X -130.6383,Y 49.3017,Z 172,A 161.0465,B 8.4643,C 0.1986,E1 8.3165,E2 290.6637} C_DIS
LIN {X -131.7905,Y 46.1341,Z 172,A 162.4878,B 8.4643,C 0.2015,E1 8.3152,E2 289.2164} C_DIS
LIN {X -132.9689,Y 42.6167,Z 172,A 163.9229,B 8.4641,C 0.2071,E1 8.3139,E2 287.7938} C_DIS
LIN {X -133.9862,Y 39.3018,Z 172,A 165.3962,B 8.4641,C 0.2103,E1 8.3127,E2 286.3155} C_DIS
LIN {X -134.9042,Y 36.0247,Z 172,A 166.8391,B 8.4639,C 0.2135,E1 8.3117,E2 284.8682} C_DIS
LIN {X -135.6717,Y 33.0184,Z 172,A 168.1446,B 8.4639,C 0.2165,E1 8.3108,E2 283.5598} C_DIS
LIN {X -136.4266,Y 29.7457,Z 172,A 169.5884,B 8.4638,C 0.2194,E1 8.3099,E2 282.109} C_DIS
LIN {X -137.2833,Y 25.5037,Z 172,A 171.3063,B 8.4636,C 0.2254,E1 8.309,E2 280.4003} C_DIS
LIN {X -138.1026,Y 20.6206,Z 172,A 173.5521,B 8.4636,C 0.2279,E1 8.308,E2 278.1292} C_DIS
LIN {X -138.6696,Y 16.3636,Z 172,A 175.8617,B 8.4636,C 0.2243,E1 8.3072,E2 275.751} C_DIS
LIN {X -139.1908,Y 11.1066,Z 172,A 177.3307,B 8.4632,C 0.2416,E1 8.3069,E2 274.3738} C_DIS
LIN {X -139.5604,Y 4.508,Z 172,A -179.7522,B 8.463,C 0.2462,E1 8.3065,E2 271.4331} C_DIS
LIN {X -139.6002,Y -3.0167,Z 172,A -176.7461,B 8.4627,C 0.2565,E1 8.3065,E2 268.4404} C_DIS
LIN {X -139.373,Y -8.4963,Z 172,A -174.3401,B 8.4627,C 0.2605,E1 8.3068,E2 266.0165} C_DIS
LIN {X -138.9564,Y -13.7207,Z 172,A -171.9085,B 8.4626,C 0.2623,E1 8.3074,E2 263.5507} C_DIS
LIN {X -138.5956,Y -16.9838,Z 172,A -170.7643,B 8.4624,C 0.2693,E1 8.3078,E2 262.4337} C_DIS
LIN {X -138.017,Y -21.1734,Z 172,A -169.0417,B 8.4622,C 0.2745,E1 8.3085,E2 260.7142} C_DIS
LIN {X -137.447,Y -24.6025,Z 172,A -167.5345,B 8.4621,C 0.2772,E1 8.3092,E2 259.1978} C_DIS
LIN {X -136.5718,Y -29.0732,Z 172,A -165.6879,B 8.4619,C 0.2829,E1 8.3102,E2 257.3556} C_DIS
LIN {X -135.7929,Y -32.5158,Z 172,A -164.2541,B 8.4618,C 0.2872,E1 8.3111,E2 255.9248} C_DIS
LIN {X -134.9277,Y -35.9367,Z 172,A -162.7905,B 8.4616,C 0.2909,E1 8.3122,E2 254.4603} C_DIS
LIN {X -134.0337,Y -39.1396,Z 172,A -161.4031,B 8.4616,C 0.2943,E1 8.3132,E2 253.071} C_DIS
LIN {X -133.1215,Y -42.1393,Z 172,A -160.0711,B 8.4614,C 0.2971,E1 8.3143,E2 251.734} C_DIS
LIN {X -132.1645,Y -45.0553,Z 172,A -158.2457,B 8.4616,C 0.2915,E1 8.3161,E2 249.8365} C_DIS
LIN {X -130.627,Y -49.3318,Z 172,A -156.9,B 8.4612,C 0.3048,E1 8.3173,E2 248.5592} C_DIS
LIN {X -128.8811,Y -53.7267,Z 172,A -154.9279,B 8.461,C 0.3094,E1 8.3194,E2 246.5844} C_DIS
LIN {X -127.5764,Y -56.7559,Z 172,A -153.5062,B 8.4609,C 0.3119,E1 8.321,E2 245.1547} C_DIS
LIN {X -126.1253,Y -59.9114,Z 172,A -152.0998,B 8.4608,C 0.3159,E1 8.3226,E2 243.7517} C_DIS
LIN {X -124.5961,Y -63.0301,Z 172,A -150.6434,B 8.4606,C 0.319,E1 8.3244,E2 242.2921} C_DIS
LIN {X -122.3359,Y -67.3163,Z 172,A -148.4979,B 8.4606,C 0.3214,E1 8.3273,E2 240.1275} C_DIS
LIN {X -120.3533,Y -70.7991,Z 172,A -146.874,B 8.4604,C 0.3258,E1 8.3296,E2 238.5071} C_DIS
LIN {X -117.9355,Y -74.7578,Z 172,A -144.9185,B 8.4602,C 0.3295,E1 8.3325,E2 236.546} C_DIS
LIN {X -115.3878,Y -78.6339,Z 172,A -142.9747,B 8.4601,C 0.3333,E1 8.3355,E2 234.5978} C_DIS
LIN {X -112.8597,Y -82.2206,Z 172,A -141.159,B 8.4599,C 0.3372,E1 8.3384,E2 232.7811} C_DIS
LIN {X -110.0843,Y -85.9015,Z 172,A -139.2279,B 8.4598,C 0.3408,E1 8.3417,E2 230.8456} C_DIS
LIN {X -107.2298,Y -89.4392,Z 172,A -137.3377,B 8.4596,C 0.3444,E1 8.3451,E2 228.953} C_DIS
LIN {X -101.4283,Y -95.9676,Z 172,A -133.8419,B 8.4593,C 0.3534,E1 8.3516,E2 225.4701} C_DIS
LIN {X -99.6627,Y -97.7996,Z 172,A -132.3331,B 8.4595,C 0.3475,E1 8.3547,E2 223.9009} C_DIS
LIN {X -96.7116,Y -100.7194,Z 172,A -130.9243,B 8.4592,C 0.3559,E1 8.3574,E2 222.5312} C_DIS
LIN {X -93.3035,Y -103.8841,Z 172,A -129.0159,B 8.459,C 0.3594,E1 8.3614,E2 220.6233} C_DIS
LIN {X -89.8732,Y -106.8656,Z 172,A -127.1263,B 8.459,C 0.3623,E1 8.3654,E2 218.7309} C_DIS
LIN {X -86.2195,Y -109.8345,Z 172,A -125.4263,B 8.4586,C 0.3697,E1 8.369,E2 217.0616} C_DIS
LIN {X -82.806,Y -112.4301,Z 172,A -123.0789,B 8.4589,C 0.3623,E1 8.3745,E2 214.6377} C_DIS
LIN {X -79.4749,Y -114.8098,Z 172,A -121.7192,B 8.4585,C 0.3706,E1 8.3775,E2 213.3201} C_DIS
LIN {X -76.311,Y -116.9366,Z 172,A -120.1018,B 8.4585,C 0.372,E1 8.3813,E2 211.696} C_DIS
LIN {X -72.4294,Y -119.3794,Z 172,A -118.2348,B 8.4584,C 0.3749,E1 8.3857,E2 209.8311} C_DIS
LIN {X -68.2685,Y -121.8067,Z 172,A -115.3582,B 8.4589,C 0.3614,E1 8.393,E2 206.8359} C_DIS
LIN {X -62.0573,Y -125.0834,Z 172,A -113.2483,B 8.4582,C 0.3788,E1 8.398,E2 204.8279} C_DIS
LIN {X -58.0906,Y -126.9751,Z 172,A -111.4143,B 8.4582,C 0.3803,E1 8.4027,E2 202.9899} C_DIS
LIN {X -54.0329,Y -128.7532,Z 172,A -109.9615,B 8.4577,C 0.3888,E1 8.4063,E2 201.5847} C_DIS
LIN {X -50.8909,Y -130.0273,Z 172,A -108.3806,B 8.4578,C 0.3867,E1 8.4104,E2 199.9789} C_DIS
LIN {X -47.6358,Y -131.2548,Z 172,A -106.9828,B 8.4578,C 0.3885,E1 8.4141,E2 198.5849} C_DIS
LIN {X -44.3837,Y -132.3898,Z 172,A -105.5846,B 8.4577,C 0.3899,E1 8.4178,E2 197.1884} C_DIS
LIN {X -41.107,Y -133.4436,Z 172,A -104.0471,B 8.4577,C 0.3887,E1 8.4219,E2 195.6342} C_DIS
LIN {X -37.4376,Y -134.5191,Z 172,A -102.4701,B 8.4577,C 0.3896,E1 8.4261,E2 194.0559} C_DIS
LIN {X -30.1065,Y -136.3487,Z 172,A -99.3206,B 8.4577,C 0.3905,E1 8.4347,E2 190.8994} C_DIS
LIN {X -26.9028,Y -137.0171,Z 172,A -97.5998,B 8.458,C 0.3839,E1 8.4396,E2 189.1283} C_DIS
LIN {X -22.6702,Y -137.7793,Z 172,A -96.2263,B 8.4576,C 0.392,E1 8.4432,E2 187.8059} C_DIS
LIN {X -17.4914,Y -138.5333,Z 172,A -94.0365,B 8.4576,C 0.3918,E1 8.4493,E2 185.6098} C_DIS
LIN {X -13.4259,Y -138.9847,Z 172,A -92.4397,B 8.4576,C 0.3936,E1 8.4537,E2 184.0231} C_DIS
LIN {X -9.1837,Y -139.3307,Z 172,A -90.6172,B 8.4576,C 0.3923,E1 8.4588,E2 182.1899} C_DIS
LIN {X -5.1157,Y -139.5384,Z 172,A -88.9702,B 8.4576,C 0.3928,E1 8.4634,E2 180.5454} C_DIS
LIN {X -0.7377,Y -139.6298,Z 172,A -87.2651,B 8.4575,C 0.3944,E1 8.4681,E2 178.8516} C_DIS
LIN {X -0.7377,Y -139.6298,Z 172,A -87.2651,B 8.4575,C 0.3944,E1 8.4681,E2 178.8516} C_DIS
Enddeposition()
LIN {X 1.0166,Y -140.5358,Z 172,A -86.6166,B 8.4575,C 0.4006,E1 8.4701,E2 178.2455} C_DIS
Startdeposition()
$VEL.CP = VEL_PRINT
LIN {X -2.6418,Y -140.5164,Z 172,A -88.6445,B 8.4569,C 0.4112,E1 8.4642,E2 180.3448} C_DIS
LIN {X -6.9814,Y -140.3674,Z 172,A -90.4058,B 8.4569,C 0.411,E1 8.4593,E2 182.1057} C_DIS
LIN {X -10.4135,Y -140.1546,Z 172,A -91.8164,B 8.4569,C 0.411,E1 8.4553,E2 183.5181} C_DIS
LIN {X -13.8691,Y -139.8555,Z 172,A -93.3433,B 8.4569,C 0.413,E1 8.4511,E2 185.0603} C_DIS
LIN {X -18.3667,Y -139.3355,Z 172,A -95.1238,B 8.4569,C 0.4114,E1 8.4461,E2 186.8329} C_DIS
LIN {X -21.8506,Y -138.8322,Z 172,A -96.5451,B 8.4569,C 0.4106,E1 8.4422,E2 188.2529} C_DIS
LIN {X -26.3994,Y -138.0389,Z 172,A -98.3946,B 8.457,C 0.4093,E1 8.4371,E2 190.0987} C_DIS
LIN {X -30.1684,Y -137.2655,Z 172,A -99.9511,B 8.457,C 0.4083,E1 8.4329,E2 191.654} C_DIS
LIN {X -33.5217,Y -136.4856,Z 172,A -101.3615,B 8.457,C 0.4077,E1 8.4291,E2 193.0657} C_DIS
LIN {X -38.4173,Y -135.1891,Z 172,A -103.4446,B 8.4571,C 0.4067,E1 8.4234,E2 195.1516} C_DIS
LIN {X -42.3018,Y -134.024,Z 172,A -105.2264,B 8.4571,C 0.4078,E1 8.4186,E2 196.9505} C_DIS
LIN {X -45.9379,Y -132.8207,Z 172,A -106.7493,B 8.4571,C 0.4058,E1 8.4146,E2 198.4686} C_DIS
LIN {X -50.1719,Y -131.2823,Z 172,A -108.5065,B 8.4573,C 0.4028,E1 8.41,E2 200.2157} C_DIS
LIN {X -52.8394,Y -130.2294,Z 172,A -109.723,B 8.4573,C 0.4025,E1 8.4069,E2 201.4385} C_DIS
LIN {X -56.5997,Y -128.6421,Z 172,A -111.6449,B 8.4573,C 0.4054,E1 8.4019,E2 203.3941} C_DIS
LIN {X -60.9209,Y -126.6506,Z 172,A -113.3301,B 8.4575,C 0.3987,E1 8.3977,E2 205.0462} C_DIS
LIN {X -64.1769,Y -125.0325,Z 172,A -115.4933,B 8.457,C 0.4089,E1 8.3921,E2 207.2977} C_DIS
LIN {X -68.9942,Y -122.4417,Z 172,A -116.9991,B 8.4578,C 0.3933,E1 8.3886,E2 208.7096} C_DIS
LIN {X -71.9879,Y -120.7058,Z 172,A -118.5898,B 8.4578,C 0.3945,E1 8.3848,E2 210.3237} C_DIS
LIN {X -75.6107,Y -118.4703,Z 172,A -120.3853,B 8.4578,C 0.3931,E1 8.3805,E2 212.1269} C_DIS
LIN {X -78.9526,Y -116.2699,Z 172,A -123.1937,B 8.4569,C 0.4108,E1 8.3737,E2 215.0863} C_DIS
LIN {X -86.1184,Y -111.0665,Z 172,A -125.2129,B 8.4585,C 0.3776,E1 8.3697,E2 216.9001} C_DIS
LIN {X -89.8756,Y -108.0492,Z 172,A -127.5902,B 8.4583,C 0.3813,E1 8.3643,E2 219.3307} C_DIS
LIN {X -93.2844,Y -105.1201,Z 172,A -129.4724,B 8.4584,C 0.3788,E1 8.3604,E2 221.219} C_DIS
LIN {X -96.6729,Y -102.0127,Z 172,A -131.5305,B 8.4584,C 0.3784,E1 8.3561,E2 223.3004} C_DIS
LIN {X -99.8947,Y -98.8599,Z 172,A -133.1878,B 8.4587,C 0.3717,E1 8.3529,E2 224.9338} C_DIS
LIN {X -102.3845,Y -96.2789,Z 172,A -134.6769,B 8.4588,C 0.3692,E1 8.35,E2 226.4258} C_DIS
LIN {X -106.6202,Y -91.5659,Z 172,A -137.08,B 8.4592,C 0.3608,E1 8.3456,E2 228.8046} C_DIS
LIN {X -108.6205,Y -89.1842,Z 172,A -138.6353,B 8.4592,C 0.3629,E1 8.3428,E2 230.3967} C_DIS
LIN {X -111.4873,Y -85.5733,Z 172,A -140.51,B 8.4593,C 0.3586,E1 8.3395,E2 232.2698} C_DIS
LIN {X -114.125,Y -82.0228,Z 172,A -142.341,B 8.4595,C 0.355,E1 8.3365,E2 234.1037} C_DIS
LIN {X -116.6622,Y -78.3725,Z 172,A -144.2152,B 8.4595,C 0.3517,E1 8.3336,E2 235.9849} C_DIS
LIN {X -119.1469,Y -74.5405,Z 172,A -146.0972,B 8.4598,C 0.3476,E1 8.3307,E2 237.8686} C_DIS
LIN {X -121.3723,Y -70.8595,Z 172,A -147.8377,B 8.4599,C 0.3431,E1 8.3283,E2 239.6064} C_DIS
LIN {X -123.5448,Y -66.9997,Z 172,A -149.7213,B 8.4601,C 0.3399,E1 8.3257,E2 241.499} C_DIS
LIN {X -125.3979,Y -63.4592,Z 172,A -151.2514,B 8.4603,C 0.3342,E1 8.3238,E2 243.0153} C_DIS
LIN {X -126.9799,Y -60.2315,Z 172,A -152.7063,B 8.4604,C 0.3303,E1 8.322,E2 244.468} C_DIS
LIN {X -128.4337,Y -57.0658,Z 172,A -154.1843,B 8.4606,C 0.3275,E1 8.3203,E2 245.9525} C_DIS
LIN {X -130.0329,Y -53.3262,Z 172,A -155.8366,B 8.4607,C 0.323,E1 8.3185,E2 247.6031} C_DIS
LIN {X -131.2029,Y -50.3762,Z 172,A -157.208,B 8.4608,C 0.3208,E1 8.3171,E2 248.9835} C_DIS
LIN {X -132.854,Y -45.8418,Z 172,A -159.1449,B 8.461,C 0.315,E1 8.3153,E2 250.915} C_DIS
LIN {X -133.907,Y -42.6679,Z 172,A -160.5905,B 8.4611,C 0.3126,E1 8.314,E2 252.3702} C_DIS
LIN {X -134.9625,Y -39.2026,Z 172,A -162.0935,B 8.4612,C 0.309,E1 8.3128,E2 253.8755} C_DIS
LIN {X -135.8365,Y -36.057,Z 172,A -163.4223,B 8.4614,C 0.3053,E1 8.3119,E2 255.203} C_DIS
LIN {X -136.7013,Y -32.627,Z 172,A -164.8918,B 8.4615,C 0.3017,E1 8.3109,E2 256.6749} C_DIS
LIN {X -137.45,Y -29.3138,Z 172,A -166.2718,B 8.4616,C 0.2977,E1 8.3101,E2 258.0532} C_DIS
LIN {X -138.0633,Y -26.2717,Z 172,A -167.5946,B 8.4617,C 0.2951,E1 8.3093,E2 259.3823} C_DIS
LIN {X -138.6615,Y -22.907,Z 172,A -168.9839,B 8.4619,C 0.291,E1 8.3087,E2 260.77} C_DIS
LIN {X -139.2121,Y -19.2884,Z 172,A -170.4886,B 8.462,C 0.287,E1 8.3081,E2 262.2751} C_DIS
LIN {X -140.0434,Y -11.8145,Z 172,A -173.647,B 8.4623,C 0.2797,E1 8.3072,E2 265.4428} C_DIS
LIN {X -140.3122,Y -8.036,Z 172,A -175.6209,B 8.4622,C 0.2819,E1 8.3068,E2 267.4699} C_DIS
LIN {X -140.4805,Y -4.1254,Z 172,A -176.8751,B 8.4625,C 0.272,E1 8.3067,E2 268.6794} C_DIS
LIN {X -140.5132,Y 2.8373,Z 172,A -179.6822,B 8.4628,C 0.2633,E1 8.3067,E2 271.4799} C_DIS
LIN {X -140.1699,Y 10.2049,Z 172,A 177.2544,B 8.463,C 0.2555,E1 8.3072,E2 274.5478} C_DIS
LIN {X -139.4738,Y 17.2972,Z 172,A 174.0933,B 8.4631,C 0.2511,E1 8.3081,E2 277.7387} C_DIS
LIN {X -138.5402,Y 23.6341,Z 172,A 171.6175,B 8.4634,C 0.2415,E1 8.3091,E2 280.1948} C_DIS
LIN {X -137.3229,Y 29.9024,Z 172,A 168.9482,B 8.4636,C 0.2351,E1 8.3106,E2 282.87} C_DIS
LIN {X -136.3378,Y 34.1157,Z 172,A 167.0946,B 8.4636,C 0.2316,E1 8.3118,E2 284.7331} C_DIS
LIN {X -135.3673,Y 37.7804,Z 172,A 165.5534,B 8.4638,C 0.2271,E1 8.3129,E2 286.2722} C_DIS
LIN {X -134.2717,Y 41.5078,Z 172,A 163.9801,B 8.4639,C 0.2226,E1 8.3142,E2 287.8426} C_DIS
LIN {X -133.1341,Y 45.0263,Z 172,A 162.4643,B 8.464,C 0.2185,E1 8.3155,E2 289.3579} C_DIS
LIN {X -132.1931,Y 47.7139,Z 172,A 161.2956,B 8.4641,C 0.2155,E1 8.3166,E2 290.5264} C_DIS
LIN {X -130.8452,Y 51.2963,Z 172,A 159.6864,B 8.4642,C 0.212,E1 8.3182,E2 292.1402} C_DIS
LIN {X -129.5101,Y 54.5796,Z 172,A 158.2029,B 8.4642,C 0.2087,E1 8.3198,E2 293.6271} C_DIS
LIN {X -128.1359,Y 57.7314,Z 172,A 156.7568,B 8.4644,C 0.2057,E1 8.3215,E2 295.0774} C_DIS
LIN {X -126.6905,Y 60.8374,Z 172,A 155.3288,B 8.4644,C 0.2025,E1 8.3232,E2 296.508} C_DIS
LIN {X -124.9344,Y 64.3696,Z 172,A 153.6053,B 8.4644,C 0.2001,E1 8.3254,E2 298.2444} C_DIS
LIN {X -122.7928,Y 68.3681,Z 172,A 151.651,B 8.4646,C 0.1971,E1 8.328,E2 300.2101} C_DIS
LIN {X -120.5319,Y 72.2798,Z 172,A 149.3669,B 8.4646,C 0.1994,E1 8.3314,E2 302.5475} C_DIS
LIN {X -117.8497,Y 76.5742,Z 172,A 148.2282,B 8.465,C 0.1797,E1 8.3329,E2 303.5681} C_DIS
LIN {X -115.0743,Y 80.6859,Z 172,A 145.6999,B 8.4649,C 0.1829,E1 8.3369,E2 306.1582} C_DIS
LIN {X -112.4542,Y 84.2994,Z 172,A 143.9223,B 8.4649,C 0.178,E1 8.3399,E2 307.9287} C_DIS
LIN {X -109.7887,Y 87.742,Z 172,A 142.2338,B 8.4651,C 0.1725,E1 8.3428,E2 309.6045} C_DIS
LIN {X -105.2043,Y 93.1891,Z 172,A 138.6983,B 8.4651,C 0.1762,E1 8.3493,E2 313.2163} C_DIS
LIN {X -101.9936,Y 96.6932,Z 172,A 137.2287,B 8.4653,C 0.1646,E1 8.352,E2 314.6257} C_DIS
LIN {X -99.4364,Y 99.3211,Z 172,A 135.1015,B 8.4651,C 0.1717,E1 8.3564,E2 316.8303} C_DIS
LIN {X -95.5643,Y 103.0519,Z 172,A 133.7976,B 8.4655,C 0.1529,E1 8.3588,E2 318.0212} C_DIS
LIN {X -90.7572,Y 107.3099,Z 172,A 130.7949,B 8.4655,C 0.1542,E1 8.3652,E2 321.07} C_DIS
LIN {X -84.8611,Y 112.0303,Z 172,A 127.3475,B 8.4655,C 0.1547,E1 8.3729,E2 324.5605} C_DIS
LIN {X -81.5082,Y 114.493,Z 172,A 126.0619,B 8.4656,C 0.145,E1 8.3757,E2 325.7933} C_DIS
LIN {X -78.1736,Y 116.7949,Z 172,A 124.3208,B 8.4656,C 0.1438,E1 8.3797,E2 327.5443} C_DIS
LIN {X -74.4614,Y 119.1961,Z 172,A 122.4768,B 8.4656,C 0.1416,E1 8.3841,E2 329.3918} C_DIS
LIN {X -70.4234,Y 121.6252,Z 172,A 120.4547,B 8.4656,C 0.1405,E1 8.389,E2 331.4249} C_DIS
LIN {X -66.6773,Y 123.7188,Z 172,A 118.7889,B 8.4657,C 0.1366,E1 8.393,E2 333.0788} C_DIS
LIN {X -62.9425,Y 125.6605,Z 172,A 117.0214,B 8.4657,C 0.1352,E1 8.3974,E2 334.8514} C_DIS
LIN {X -57.4868,Y 128.2454,Z 172,A 114.9501,B 8.4659,C 0.1254,E1 8.4025,E2 336.8718} C_DIS
LIN {X -53.7648,Y 129.8504,Z 172,A 113.0144,B 8.4659,C 0.1284,E1 8.4076,E2 338.8418} C_DIS
LIN {X -50.3418,Y 131.2162,Z 172,A 110.7218,B 8.4657,C 0.1405,E1 8.4138,E2 341.2316} C_DIS
LIN {X -44.7392,Y 133.2297,Z 172,A 109.2435,B 8.466,C 0.1217,E1 8.4174,E2 342.59} C_DIS
LIN {X -41.7657,Y 134.1928,Z 172,A 107.683,B 8.466,C 0.1256,E1 8.4217,E2 344.1856} C_DIS
LIN {X -37.7664,Y 135.3712,Z 172,A 106.0413,B 8.466,C 0.1231,E1 8.426,E2 345.8188} C_DIS
LIN {X -33.7508,Y 136.4301,Z 172,A 104.3881,B 8.466,C 0.1212,E1 8.4305,E2 347.4659} C_DIS
LIN {X -30.0702,Y 137.2867,Z 172,A 102.4159,B 8.4659,C 0.1279,E1 8.436,E2 349.491} C_DIS
LIN {X -26.2264,Y 138.072,Z 172,A 100.939,B 8.4659,C 0.1248,E1 8.44,E2 350.9516} C_DIS
LIN {X -23.0225,Y 138.6422,Z 172,A 99.6766,B 8.4659,C 0.123,E1 8.4435,E2 352.2052} C_DIS
LIN {X -18.1684,Y 139.3615,Z 172,A 97.8873,B 8.466,C 0.1183,E1 8.4483,E2 353.967} C_DIS
LIN {X -14.7548,Y 139.7644,Z 172,A 96.4507,B 8.466,C 0.1185,E1 8.4523,E2 355.4072} C_DIS
LIN {X -10.651,Y 140.1373,Z 172,A 94.9546,B 8.466,C 0.1147,E1 8.4564,E2 356.8794} C_DIS
LIN {X -8.0117,Y 140.3137,Z 172,A 93.7368,B 8.466,C 0.1171,E1 8.4599,E2 358.1142} C_DIS
LIN {X -3.6278,Y 140.4944,Z 172,A 91.873,B 8.466,C 0.1182,E1 8.4651,E2 359.9865} C_DIS
LIN {X 0.4149,Y 140.5408,Z 172,A 90.1791,B 8.466,C 0.119,E1 8.4699,E2 361.6853} C_DIS
LIN {X 3.9513,Y 140.4854,Z 172,A 88.7953,B 8.466,C 0.118,E1 8.4737,E2 363.0612} C_DIS
LIN {X 7.582,Y 140.3372,Z 172,A 87.3959,B 8.466,C 0.1167,E1 8.4776,E2 364.4498} C_DIS
LIN {X 10.25,Y 140.1666,Z 172,A 86.2124,B 8.466,C 0.1186,E1 8.4809,E2 365.6446} C_DIS
LIN {X 13.7596,Y 139.866,Z 172,A 84.8264,B 8.466,C 0.1181,E1 8.4847,E2 367.0237} C_DIS
LIN {X 17.21,Y 139.4842,Z 172,A 83.4649,B 8.466,C 0.1175,E1 8.4885,E2 368.3781} C_DIS
LIN {X 20.8829,Y 138.982,Z 172,A 81.711,B 8.466,C 0.1227,E1 8.4934,E2 370.1619} C_DIS
LIN {X 25.032,Y 138.2937,Z 172,A 80.23,B 8.466,C 0.1191,E1 8.4974,E2 371.6131} C_DIS
LIN {X 28.4611,Y 137.6293,Z 172,A 78.6484,B 8.466,C 0.1229,E1 8.5018,E2 373.2141} C_DIS
LIN {X 35.1013,Y 136.0876,Z 172,A 76.0808,B 8.466,C 0.1206,E1 8.5087,E2 375.7546} C_DIS
LIN {X 37.717,Y 135.385,Z 172,A 74.8477,B 8.466,C 0.124,E1 8.5121,E2 377.0036} C_DIS
LIN {X 42.007,Y 134.1181,Z 172,A 72.9745,B 8.466,C 0.1264,E1 8.5171,E2 378.8828} C_DIS
LIN {X 46.1138,Y 132.7597,Z 172,A 71.3343,B 8.466,C 0.1256,E1 8.5214,E2 380.5071} C_DIS
LIN {X 49.36,Y 131.5873,Z 172,A 69.8945,B 8.4659,C 0.1277,E1 8.5252,E2 381.9508} C_DIS
LIN {X 53.4533,Y 129.9805,Z 172,A 67.9488,B 8.4659,C 0.1326,E1 8.5303,E2 383.9157} C_DIS
LIN {X 57.7867,Y 128.1112,Z 172,A 66.2411,B 8.4659,C 0.1305,E1 8.5345,E2 385.5961} C_DIS
LIN {X 60.973,Y 126.6257,Z 172,A 64.8103,B 8.4659,C 0.1322,E1 8.5382,E2 387.0265} C_DIS
LIN {X 66.5328,Y 123.7964,Z 172,A 62.2255,B 8.4658,C 0.1364,E1 8.5446,E2 389.6167} C_DIS
LIN {X 70.4274,Y 121.6229,Z 172,A 60.4356,B 8.4658,C 0.1384,E1 8.5489,E2 391.4031} C_DIS
LIN {X 74.616,Y 119.0999,Z 172,A 58.6771,B 8.4658,C 0.1366,E1 8.553,E2 393.1321} C_DIS
LIN {X 77.3724,Y 117.3272,Z 172,A 57.143,B 8.4656,C 0.1427,E1 8.5567,E2 394.6914} C_DIS
LIN {X 83.5776,Y 112.9917,Z 172,A 54.2996,B 8.4656,C 0.1428,E1 8.5631,E2 397.5047} C_DIS
LIN {X 87.688,Y 109.8317,Z 172,A 51.9941,B 8.4656,C 0.1505,E1 8.5683,E2 399.8348} C_DIS
LIN {X 91.0378,Y 107.0713,Z 172,A 50.2125,B 8.4655,C 0.154,E1 8.5721,E2 401.6184} C_DIS
LIN {X 94.5854,Y 103.9509,Z 172,A 48.2722,B 8.4654,C 0.158,E1 8.5761,E2 403.5609} C_DIS
LIN {X 97.9712,Y 100.7664,Z 172,A 46.557,B 8.4654,C 0.158,E1 8.5795,E2 405.2539} C_DIS
LIN {X 100.5755,Y 98.1674,Z 172,A 44.9448,B 8.4653,C 0.1634,E1 8.5827,E2 406.8809} C_DIS
LIN {X 103.6295,Y 94.9375,Z 172,A 43.0772,B 8.4652,C 0.1683,E1 8.5863,E2 408.7561} C_DIS
LIN {X 106.9061,Y 91.2321,Z 172,A 41.1548,B 8.4652,C 0.1707,E1 8.5898,E2 410.6674} C_DIS
LIN {X 110.0414,Y 87.4245,Z 172,A 39.37,B 8.4652,C 0.1704,E1 8.5929,E2 412.4242} C_DIS
LIN {X 112.1044,Y 84.763,Z 172,A 37.8746,B 8.465,C 0.1761,E1 8.5955,E2 413.9359} C_DIS
LIN {X 114.6596,Y 81.2738,Z 172,A 36.0795,B 8.465,C 0.1809,E1 8.5984,E2 415.7358} C_DIS
LIN {X 117.5289,Y 77.0661,Z 172,A 34.2875,B 8.465,C 0.1798,E1 8.6011,E2 417.4926} C_DIS
LIN {X 119.2352,Y 74.3986,Z 172,A 32.3267,B 8.4646,C 0.1972,E1 8.6042,E2 419.5393} C_DIS
LIN {X 121.6987,Y 70.2965,Z 172,A 30.956,B 8.4647,C 0.1897,E1 8.606,E2 420.8374} C_DIS
LIN {X 123.6164,Y 66.8677,Z 172,A 29.2585,B 8.4646,C 0.1958,E1 8.6083,E2 422.5481} C_DIS
LIN {X 125.4284,Y 63.3992,Z 172,A 27.8026,B 8.4646,C 0.1968,E1 8.6101,E2 423.987} C_DIS
LIN {X 127.2351,Y 59.6945,Z 172,A 26.175,B 8.4645,C 0.2,E1 8.6121,E2 425.609} C_DIS
LIN {X 128.3859,Y 57.1727,Z 172,A 25.0076,B 8.4645,C 0.2038,E1 8.6135,E2 426.7819} C_DIS
LIN {X 130.504,Y 52.1584,Z 172,A 22.8846,B 8.4643,C 0.2076,E1 8.6157,E2 428.894} C_DIS
LIN {X 131.6505,Y 49.1911,Z 172,A 21.5896,B 8.4643,C 0.2111,E1 8.617,E2 430.1897} C_DIS
LIN {X 132.736,Y 46.1823,Z 172,A 20.2335,B 8.4641,C 0.2157,E1 8.6183,E2 431.5533} C_DIS
LIN {X 133.9577,Y 42.5091,Z 172,A 18.7295,B 8.4641,C 0.2184,E1 8.6196,E2 433.049} C_DIS
LIN {X 134.9761,Y 39.1563,Z 172,A 17.3372,B 8.464,C 0.2216,E1 8.6207,E2 434.4376} C_DIS
LIN {X 135.9804,Y 35.5176,Z 172,A 15.8263,B 8.4639,C 0.2253,E1 8.6218,E2 435.9462} C_DIS
LIN {X 137.1865,Y 30.5312,Z 172,A 13.775,B 8.4637,C 0.2303,E1 8.6231,E2 437.994} C_DIS
LIN {X 137.8296,Y 27.4772,Z 172,A 12.5223,B 8.4637,C 0.2334,E1 8.6238,E2 439.2451} C_DIS
LIN {X 138.3809,Y 24.5451,Z 172,A 11.3146,B 8.4636,C 0.2367,E1 8.6244,E2 440.4527} C_DIS
LIN {X 139.0425,Y 20.4756,Z 172,A 9.2465,B 8.4632,C 0.25,E1 8.6253,E2 442.5719} C_DIS
LIN {X 139.5655,Y 16.5288,Z 172,A 8.0525,B 8.4633,C 0.2452,E1 8.6257,E2 443.7122} C_DIS
LIN {X 139.9066,Y 13.3365,Z 172,A 6.7354,B 8.4633,C 0.2491,E1 8.626,E2 445.0314} C_DIS
LIN {X 140.2318,Y 9.3423,Z 172,A 5.0513,B 8.463,C 0.255,E1 8.6264,E2 446.7235} C_DIS
LIN {X 140.4424,Y 5.2648,Z 172,A 3.5186,B 8.463,C 0.2569,E1 8.6266,E2 448.2407} C_DIS
LIN {X 140.5377,Y 1.1009,Z 172,A 1.7782,B 8.4628,C 0.2627,E1 8.6266,E2 449.9881} C_DIS
LIN {X 140.507,Y -3.1741,Z 172,A 0.2017,B 8.4628,C 0.2641,E1 8.6266,E2 451.5448} C_DIS
LIN {X 140.3788,Y -6.7543,Z 172,A -1.4043,B 8.4625,C 0.2715,E1 8.6264,E2 453.1709} C_DIS
LIN {X 140.0704,Y -11.4939,Z 172,A -3.1931,B 8.4625,C 0.2739,E1 8.626,E2 454.9424} C_DIS
LIN {X 139.703,Y -15.3258,Z 172,A -4.7248,B 8.4623,C 0.2776,E1 8.6256,E2 456.4707} C_DIS
LIN {X 139.3345,Y -18.3743,Z 172,A -5.9986,B 8.4622,C 0.2817,E1 8.6252,E2 457.7485} C_DIS
LIN {X 138.7656,Y -22.2789,Z 172,A -7.6934,B 8.462,C 0.2882,E1 8.6244,E2 459.4562} C_DIS
LIN {X 137.9843,Y -26.6849,Z 172,A -9.6221,B 8.4617,C 0.2957,E1 8.6234,E2 461.4} C_DIS
LIN {X 137.3056,Y -29.9826,Z 172,A -10.6443,B 8.4618,C 0.2919,E1 8.6229,E2 462.3782} C_DIS
LIN {X 135.9191,Y -35.7474,Z 172,A -12.9229,B 8.4618,C 0.2957,E1 8.6214,E2 464.6413} C_DIS
LIN {X 134.3469,Y -41.2621,Z 172,A -15.3994,B 8.4614,C 0.3053,E1 8.6194,E2 467.1383} C_DIS
LIN {X 133.0407,Y -45.3034,Z 172,A -17.0813,B 8.4612,C 0.309,E1 8.6179,E2 468.8156} C_DIS
LIN {X 131.4529,Y -49.7186,Z 172,A -18.9643,B 8.4611,C 0.3136,E1 8.6161,E2 470.6966} C_DIS
LIN {X 130.0229,Y -53.3514,Z 172,A -20.5067,B 8.461,C 0.3169,E1 8.6145,E2 472.2343} C_DIS
LIN {X 128.7019,Y -56.4622,Z 172,A -21.9724,B 8.4607,C 0.3225,E1 8.6129,E2 473.7128} C_DIS
LIN {X 126.8165,Y -60.5736,Z 172,A -23.587,B 8.4607,C 0.3224,E1 8.611,E2 475.2993} C_DIS
LIN {X 124.3252,Y -65.5353,Z 172,A -25.5377,B 8.4607,C 0.3215,E1 8.6087,E2 477.2114} C_DIS
LIN {X 122.8547,Y -68.2562,Z 172,A -27.2233,B 8.4603,C 0.3341,E1 8.6063,E2 478.9541} C_DIS
LIN {X 120.8382,Y -71.7659,Z 172,A -28.8627,B 8.4601,C 0.338,E1 8.604,E2 480.5938} C_DIS
LIN {X 117.3235,Y -77.378,Z 172,A -31.2742,B 8.4601,C 0.3385,E1 8.6005,E2 482.9703} C_DIS
LIN {X 113.6142,Y -82.7288,Z 172,A -34.3847,B 8.4595,C 0.3549,E1 8.5953,E2 486.1432} C_DIS
LIN {X 111.4576,Y -85.612,Z 172,A -35.6809,B 8.4595,C 0.3546,E1 8.5932,E2 487.4186} C_DIS
LIN {X 108.369,Y -89.4893,Z 172,A -37.5762,B 8.4594,C 0.3566,E1 8.5899,E2 489.2995} C_DIS
LIN {X 105.5696,Y -92.776,Z 172,A -39.3518,B 8.4592,C 0.3609,E1 8.5866,E2 491.079} C_DIS
LIN {X 102.17,Y -96.5062,Z 172,A -41.2582,B 8.4592,C 0.3622,E1 8.583,E2 492.9675} C_DIS
LIN {X 100.3465,Y -98.4009,Z 172,A -42.3934,B 8.459,C 0.3658,E1 8.5808,E2 494.1121} C_DIS
LIN {X 97.2309,Y -101.4807,Z 172,A -44.1353,B 8.4589,C 0.3686,E1 8.5773,E2 495.85} C_DIS
LIN {X 94.0531,Y -104.4333,Z 172,A -45.9575,B 8.4587,C 0.3734,E1 8.5736,E2 497.6809} C_DIS
LIN {X 90.8688,Y -107.215,Z 172,A -47.4743,B 8.4587,C 0.3724,E1 8.5704,E2 499.1723} C_DIS
LIN {X 88.2252,Y -109.4005,Z 172,A -48.9848,B 8.4585,C 0.3774,E1 8.5671,E2 500.6987} C_DIS
LIN {X 84.6617,Y -112.1809,Z 172,A -50.8146,B 8.4583,C 0.3806,E1 8.563,E2 502.5286} C_DIS
LIN {X 81.001,Y -114.8521,Z 172,A -52.8252,B 8.458,C 0.3873,E1 8.5584,E2 504.5623} C_DIS
LIN {X 78.3387,Y -116.6848,Z 172,A -53.8806,B 8.4582,C 0.384,E1 8.5561,E2 505.5846} C_DIS
LIN {X 74.8769,Y -118.9354,Z 172,A -55.6841,B 8.458,C 0.3893,E1 8.5518,E2 507.4052} C_DIS
LIN {X 68.8564,Y -122.5192,Z 172,A -58.45,B 8.4578,C 0.3919,E1 8.5451,E2 510.1618} C_DIS
LIN {X 65.0589,Y -124.5753,Z 172,A -60.1614,B 8.4578,C 0.3934,E1 8.5409,E2 511.8682} C_DIS
LIN {X 60.2206,Y -126.9851,Z 172,A -63.1052,B 8.4569,C 0.4117,E1 8.5333,E2 514.9101} C_DIS
LIN {X 54.5159,Y -129.5367,Z 172,A -64.6533,B 8.4577,C 0.3944,E1 8.5296,E2 516.3299} C_DIS
LIN {X 51.9697,Y -130.58,Z 172,A -65.9237,B 8.4575,C 0.3988,E1 8.5263,E2 517.6209} C_DIS
LIN {X 48.9058,Y -131.7574,Z 172,A -67.3105,B 8.4574,C 0.4013,E1 8.5226,E2 519.015} C_DIS
LIN {X 45.0228,Y -133.1353,Z 172,A -69.1383,B 8.4572,C 0.4061,E1 8.5178,E2 520.8635} C_DIS
LIN {X 40.8186,Y -134.4826,Z 172,A -70.7526,B 8.4572,C 0.4041,E1 8.5135,E2 522.4547} C_DIS
LIN {X 36.8934,Y -135.6135,Z 172,A -72.6447,B 8.457,C 0.4102,E1 8.5083,E2 524.3778} C_DIS
LIN {X 33.7454,Y -136.4316,Z 172,A -73.6904,B 8.4572,C 0.4056,E1 8.5056,E2 525.3877} C_DIS
LIN {X 31.2093,Y -137.0316,Z 172,A -74.776,B 8.4572,C 0.4069,E1 8.5026,E2 526.477} C_DIS
LIN {X 27.5536,Y -137.814,Z 172,A -76.2621,B 8.4572,C 0.4072,E1 8.4986,E2 527.9591} C_DIS
LIN {X 24.5142,Y -138.3864,Z 172,A -77.5226,B 8.4571,C 0.408,E1 8.4951,E2 529.2203} C_DIS
LIN {X 19.1771,Y -139.2279,Z 172,A -79.7081,B 8.4571,C 0.4089,E1 8.4891,E2 531.405} C_DIS
LIN {X 16.125,Y -139.6136,Z 172,A -80.9774,B 8.457,C 0.4098,E1 8.4856,E2 532.677} C_DIS
LIN {X 11.975,Y -140.0298,Z 172,A -82.7115,B 8.457,C 0.4111,E1 8.4807,E2 534.4164} C_DIS
LIN {X 7.9977,Y -140.3146,Z 172,A -84.2756,B 8.457,C 0.4104,E1 8.4764,E2 535.9734} C_DIS
LIN {X 4.367,Y -140.4738,Z 172,A -85.8169,B 8.4569,C 0.4119,E1 8.4721,E2 537.5233} C_DIS
LIN {X 1.0166,Y -140.5358,Z 172,A -86.6136,B 8.4574,C 0.4011,E1 8.4701,E2 538.2456} C_DIS
Enddeposition()
LIN {X 1.0166,Y -140.5358,Z 172,A -86.6136,B 8.4574,C 0.4011,E1 8.4701,E2 538.2456} C_DIS
Startdeposition()
$VEL.CP = VEL_PRINT
LIN {X 1.7352,Y -141.4408,Z 172,A -86.1834,B 8.4573,C 0.4032,E1 8.4712,E2 537.8303} C_DIS
LIN {X 5.2114,Y -141.3543,Z 172,A -84.7875,B 8.4573,C 0.4032,E1 8.4751,E2 536.4353} C_DIS
LIN {X 8.6858,Y -141.1831,Z 172,A -83.3183,B 8.4573,C 0.4016,E1 8.4792,E2 534.9573} C_DIS
LIN {X 13.2188,Y -140.8313,Z 172,A -81.445,B 8.4574,C 0.4002,E1 8.4844,E2 533.0788} C_DIS
LIN {X 17.985,Y -140.3024,Z 172,A -79.6082,B 8.4574,C 0.4015,E1 8.4895,E2 531.255} C_DIS
LIN {X 20.7784,Y -139.9176,Z 172,A -78.4802,B 8.4574,C 0.4012,E1 8.4926,E2 530.1283} C_DIS
LIN {X 24.1994,Y -139.3663,Z 172,A -77.0689,B 8.4574,C 0.4002,E1 8.4965,E2 528.7151} C_DIS
LIN {X 27.6034,Y -138.7316,Z 172,A -75.6757,B 8.4574,C 0.3994,E1 8.5003,E2 527.3222} C_DIS
LIN {X 30.9882,Y -138.0146,Z 172,A -74.2822,B 8.4575,C 0.3985,E1 8.5041,E2 525.9288} C_DIS
LIN {X 34.9884,Y -137.0543,Z 172,A -72.5813,B 8.4576,C 0.3965,E1 8.5087,E2 524.2222} C_DIS
LIN {X 39.3991,Y -135.8523,Z 172,A -70.7842,B 8.4576,C 0.3959,E1 8.5136,E2 522.4311} C_DIS
LIN {X 42.7401,Y -134.8384,Z 172,A -69.3792,B 8.4576,C 0.3948,E1 8.5173,E2 521.0263} C_DIS
LIN {X 46.6413,Y -133.5391,Z 172,A -67.7235,B 8.4578,C 0.3932,E1 8.5217,E2 519.3706} C_DIS
LIN {X 49.9003,Y -132.3557,Z 172,A -66.3053,B 8.4578,C 0.3914,E1 8.5254,E2 517.9496} C_DIS
LIN {X 53.5288,Y -130.9318,Z 172,A -64.6145,B 8.458,C 0.3872,E1 8.5298,E2 516.2426} C_DIS
LIN {X 57.6423,Y -129.1718,Z 172,A -62.9657,B 8.458,C 0.3883,E1 8.534,E2 514.6142} C_DIS
LIN {X 60.7712,Y -127.7297,Z 172,A -61.5378,B 8.458,C 0.3857,E1 8.5376,E2 513.1808} C_DIS
LIN {X 63.8901,Y -126.1987,Z 172,A -60.1858,B 8.4581,C 0.3849,E1 8.541,E2 511.8351} C_DIS
LIN {X 66.9731,Y -124.5919,Z 172,A -58.694,B 8.4583,C 0.3811,E1 8.5447,E2 510.3309} C_DIS
LIN {X 70.972,Y -122.3582,Z 172,A -56.9014,B 8.4583,C 0.3796,E1 8.549,E2 508.5452} C_DIS
LIN {X 74.6807,Y -120.1305,Z 172,A -55.1098,B 8.4585,C 0.376,E1 8.5533,E2 506.7467} C_DIS
LIN {X 78.5853,Y -117.6133,Z 172,A -53.26,B 8.4586,C 0.3735,E1 8.5576,E2 504.8996} C_DIS
LIN {X 82.1702,Y -115.1373,Z 172,A -51.5143,B 8.4588,C 0.3708,E1 8.5616,E2 503.1548} C_DIS
LIN {X 85.6577,Y -112.5673,Z 172,A -49.7628,B 8.4588,C 0.3677,E1 8.5655,E2 501.4021} C_DIS
LIN {X 89.0645,Y -109.8915,Z 172,A -48.0746,B 8.459,C 0.3658,E1 8.5692,E2 499.7211} C_DIS
LIN {X 92.4039,Y -107.0983,Z 172,A -46.3014,B 8.4591,C 0.3621,E1 8.573,E2 497.945} C_DIS
LIN {X 95.8803,Y -103.9977,Z 172,A -44.4306,B 8.4593,C 0.3586,E1 8.5768,E2 496.0745} C_DIS
LIN {X 99.1751,Y -100.8606,Z 172,A -42.6582,B 8.4593,C 0.3563,E1 8.5804,E2 494.3098} C_DIS
LIN {X 102.0838,Y -97.9157,Z 172,A -40.9506,B 8.4596,C 0.352,E1 8.5837,E2 492.5963} C_DIS
LIN {X 105.0352,Y -94.7433,Z 172,A -39.2076,B 8.4597,C 0.3484,E1 8.587,E2 490.8533} C_DIS
LIN {X 108.0271,Y -91.3171,Z 172,A -37.3727,B 8.4599,C 0.3444,E1 8.5903,E2 489.0175} C_DIS
LIN {X 111.0099,Y -87.6667,Z 172,A -35.548,B 8.4599,C 0.3419,E1 8.5935,E2 487.2022} C_DIS
LIN {X 113.6419,Y -84.2268,Z 172,A -33.8331,B 8.4601,C 0.3386,E1 8.5964,E2 485.4908} C_DIS
LIN {X 116.1599,Y -80.718,Z 172,A -32.0781,B 8.4603,C 0.3342,E1 8.5992,E2 483.7332} C_DIS
LIN {X 118.5635,Y -77.1443,Z 172,A -30.3853,B 8.4603,C 0.331,E1 8.6018,E2 482.0456} C_DIS
LIN {X 120.8799,Y -73.4621,Z 172,A -28.605,B 8.4606,C 0.3262,E1 8.6044,E2 480.261} C_DIS
LIN {X 123.0739,Y -69.7246,Z 172,A -26.8667,B 8.4607,C 0.3221,E1 8.6069,E2 478.5232} C_DIS
LIN {X 125.0637,Y -66.0845,Z 172,A -25.3306,B 8.4607,C 0.321,E1 8.6089,E2 477.0045} C_DIS
LIN {X 126.5269,Y -63.2412,Z 172,A -23.9221,B 8.461,C 0.315,E1 8.6107,E2 475.5796} C_DIS
LIN {X 128.2447,Y -59.6772,Z 172,A -22.4731,B 8.461,C 0.3142,E1 8.6124,E2 474.1494} C_DIS
LIN {X 129.752,Y -56.3242,Z 172,A -21.1353,B 8.461,C 0.3136,E1 8.6139,E2 472.8301} C_DIS
LIN {X 130.9317,Y -53.5289,Z 172,A -19.6867,B 8.4614,C 0.3053,E1 8.6154,E2 471.3511} C_DIS
LIN {X 132.5819,Y -49.2965,Z 172,A -17.9812,B 8.4614,C 0.3033,E1 8.6171,E2 469.6616} C_DIS
LIN {X 133.7574,Y -46.0116,Z 172,A -16.5119,B 8.4616,C 0.2982,E1 8.6185,E2 468.1834} C_DIS
LIN {X 135.181,Y -41.6434,Z 172,A -14.8974,B 8.4616,C 0.2985,E1 8.6198,E2 466.5997} C_DIS
LIN {X 136.0418,Y -38.744,Z 172,A -13.556,B 8.4618,C 0.2925,E1 8.6209,E2 465.2417} C_DIS
LIN {X 137.0569,Y -34.9779,Z 172,A -12.0052,B 8.4619,C 0.2887,E1 8.622,E2 463.6932} C_DIS
LIN {X 137.7741,Y -32.0411,Z 172,A -10.7979,B 8.462,C 0.2856,E1 8.6228,E2 462.487} C_DIS
LIN {X 138.5198,Y -28.6446,Z 172,A -9.4109,B 8.4622,C 0.282,E1 8.6236,E2 461.1014} C_DIS
LIN {X 139.1803,Y -25.2391,Z 172,A -8.2247,B 8.4622,C 0.283,E1 8.6242,E2 459.9427} C_DIS
LIN {X 139.6573,Y -22.4626,Z 172,A -6.902,B 8.4624,C 0.2756,E1 8.6248,E2 458.595} C_DIS
LIN {X 140.1651,Y -19.0329,Z 172,A -5.5207,B 8.4624,C 0.2721,E1 8.6253,E2 457.2154} C_DIS
LIN {X 140.5885,Y -15.5935,Z 172,A -4.029,B 8.4627,C 0.266,E1 8.6258,E2 455.7106} C_DIS
LIN {X 141.0194,Y -11.0547,Z 172,A -2.1805,B 8.4628,C 0.2607,E1 8.6263,E2 453.8602} C_DIS
LIN {X 141.2802,Y -6.9323,Z 172,A -0.6055,B 8.4629,C 0.258,E1 8.6265,E2 452.2965} C_DIS
LIN {X 141.4278,Y -2.5179,Z 172,A 1.0903,B 8.463,C 0.2549,E1 8.6266,E2 450.6114} C_DIS
LIN {X 141.4409,Y 1.7301,Z 172,A 2.7812,B 8.4631,C 0.2506,E1 8.6266,E2 448.923} C_DIS
LIN {X 141.3541,Y 5.2182,Z 172,A 4.1539,B 8.4632,C 0.2475,E1 8.6265,E2 447.5543} C_DIS
LIN {X 141.1834,Y 8.6799,Z 172,A 5.5991,B 8.4634,C 0.2425,E1 8.6262,E2 446.1024} C_DIS
LIN {X 140.8317,Y 13.214,Z 172,A 7.449,B 8.4635,C 0.237,E1 8.6258,E2 444.2499} C_DIS
LIN {X 140.3029,Y 17.9817,Z 172,A 9.2552,B 8.4635,C 0.2345,E1 8.6252,E2 442.46} C_DIS
LIN {X 139.9184,Y 20.7723,Z 172,A 10.3643,B 8.4637,C 0.232,E1 8.6248,E2 441.3542} C_DIS
LIN {X 139.3681,Y 24.1896,Z 172,A 11.7575,B 8.4637,C 0.2282,E1 8.6241,E2 439.9611} C_DIS
LIN {X 138.7343,Y 27.5903,Z 172,A 13.1319,B 8.4639,C 0.2248,E1 8.6234,E2 438.5891} C_DIS
LIN {X 138.018,Y 30.9737,Z 172,A 14.5079,B 8.4639,C 0.2214,E1 8.6226,E2 437.2151} C_DIS
LIN {X 137.0512,Y 35.0004,Z 172,A 16.1974,B 8.4641,C 0.2164,E1 8.6215,E2 435.5228} C_DIS
LIN {X 135.894,Y 39.2566,Z 172,A 17.9517,B 8.4641,C 0.2122,E1 8.6201,E2 433.7713} C_DIS
LIN {X 134.8442,Y 42.7217,Z 172,A 19.3547,B 8.4642,C 0.2096,E1 8.619,E2 432.3756} C_DIS
LIN {X 133.5428,Y 46.6305,Z 172,A 20.997,B 8.4643,C 0.2056,E1 8.6175,E2 430.7356} C_DIS
LIN {X 132.357,Y 49.897,Z 172,A 22.4177,B 8.4644,C 0.2015,E1 8.6161,E2 429.3122} C_DIS
LIN {X 130.9274,Y 53.5395,Z 172,A 24.0807,B 8.4646,C 0.1956,E1 8.6144,E2 427.6379} C_DIS
LIN {X 129.3129,Y 57.3268,Z 172,A 25.6148,B 8.4646,C 0.1941,E1 8.6127,E2 426.1202} C_DIS
LIN {X 127.8739,Y 60.4694,Z 172,A 26.9607,B 8.4646,C 0.1917,E1 8.6111,E2 424.7805} C_DIS
LIN {X 126.1987,Y 63.8901,Z 172,A 28.4776,B 8.4647,C 0.1883,E1 8.6092,E2 423.266} C_DIS
LIN {X 124.3389,Y 67.4424,Z 172,A 30.1845,B 8.4649,C 0.1823,E1 8.607,E2 421.5475} C_DIS
LIN {X 122.1984,Y 71.248,Z 172,A 31.9329,B 8.4649,C 0.1784,E1 8.6045,E2 419.8007} C_DIS
LIN {X 119.9367,Y 74.992,Z 172,A 33.6108,B 8.465,C 0.1761,E1 8.6021,E2 418.1341} C_DIS
LIN {X 117.6179,Y 78.5784,Z 172,A 35.3621,B 8.465,C 0.1715,E1 8.5994,E2 416.3791} C_DIS
Enddeposition()
END
